			bBusy				=> xReadBusy,
			bError				=> xError,
			nErrID				=> udiErrID,
			iErrPos				=> usiErrPos,
			stMDP_DynAddr		=> ,
			iModuleTypeCount	=> ,
			iModuleCount		=> ,
			stMDP_ModuleHeader	=> ,
			arrStartIdx			=> ,
		);
	ELSE
		fbMDP_ReadModule(
			bExecute			:= FALSE,

			bBusy				=> xReadBusy,
			bError				=> xError,
			nErrID 				=> udiErrID,
			iErrPos				=> usiErrPos,
		);
		IF NOT xReadBusy THEN
			// allocate received module header
			stMDP_ModuleHeader	:= fbMDP_ReadModule.stMDP_ModuleHeader;
			// allocate information of startindexes in data buffer
			MEMCPY(ADR(arrStartIdx), ADR(fbMDP_ReadModule.arrStartIdx), SIZEOF(arrStartIdx) );
			// reset module content struct
			MEMSET( ADR(stMDP_ModuleContent), 0, SIZEOF(stMDP_ModuleContent) );
			// allocate received data to DiskMngmntTBL4 struct
			stMDP_ModuleContent.uiLen		:= arrData[0];
			MEMCPY(ADR(stMDP_ModuleContent.udiDriveType1), 	ADR(arrData)+arrStartIdx[1], MIN(arrStartIdx[2]-arrStartIdx[1], SIZEOF(stMDP_ModuleContent.udiDriveType1)) );
			MEMCPY(ADR(stMDP_ModuleContent.udiDriveType2), 	ADR(arrData)+arrStartIdx[2], MIN(arrStartIdx[3]-arrStartIdx[2], SIZEOF(stMDP_ModuleContent.udiDriveType2))  );
			MEMCPY(ADR(stMDP_ModuleContent.udiDriveType3), 	ADR(arrData)+arrStartIdx[3], MIN(arrStartIdx[4]-arrStartIdx[3], SIZEOF(stMDP_ModuleContent.udiDriveType3)) );
			MEMCPY(ADR(stMDP_ModuleContent.udiDriveType4), 	ADR(arrData)+arrStartIdx[4], MIN(arrStartIdx[5]-arrStartIdx[4], SIZEOF(stMDP_ModuleContent.udiDriveType4)) );
			MEMCPY(ADR(stMDP_ModuleContent.udiDriveType5),	ADR(arrData)+arrStartIdx[5], MIN(arrStartIdx[6]-arrStartIdx[5], SIZEOF(stMDP_ModuleContent.udiDriveType5)) );
			MEMCPY(ADR(stMDP_ModuleContent.udiDriveType6),	ADR(arrData)+arrStartIdx[6], MIN(arrStartIdx[7]-arrStartIdx[6], SIZEOF(stMDP_ModuleContent.udiDriveType6)) );

			// reset FB
			xBusy 				:= FALSE;
		END_IF
	END_IF

	// check timeout
	TimeOut();
	IF TimeOut.Q THEN
		TimeOut(IN 				:= FALSE);
		xError					:= TRUE;
		udiErrID				:= INT_TO_UINT(eMDP_Err_PLC) * 16#10000 + INT_TO_UINT(eMDP_ErrPLC_TimeOut);
	END_IF
END_IF

IF xError THEN
	// reset FB
	xBusy 						:= FALSE;
END_IF

END_FUNCTION_BLOCK

// ---- POUs/Safety_Diagnostics/AX5805_ADS_Reads.TcPOU
PROGRAM AX5805_ADS_Reads
//		8-2-2012
// 		This Program has been supplied by Beckhoff Automation As-Is and is intended only as an example 
//		implementation. Functionality is not guaranteed. 
//
VAR
	//Time to check CoE values
	T1							: 		TON ;
	xExecute					: 		BOOL ;
	tTime1						: 		TIME ;

	//Counter for just some very simple sequencing
	C1							: 		CTU ;
	xReset						: 		BOOL ;
	wPreset						: 		WORD := 10 ;
	xDone						: 		BOOL ;
	wCount						: 		WORD ;

	// Reading the serial number out of the AX5805
	fbAX5805Sn_ADSRead			: 		ADSREAD ;
	dwAX5805_Sn					: 		DWORD ;
	xAX5805Sn_busy				: 		BOOL ;
	xAX5805Sn_Err				: 		BOOL ;
	xAX5805Sn_ErrID				: 		UDINT ;

	// Reading the DIP Switch Setting out of the AX5805
	fbAX5805DSw_ADSRead			: 		ADSREAD ;
	wAX5805_DSw					: 		WORD ;
	xAX5805DSw_busy				: 		BOOL ;
	xAX5805DSw_Err				: 		BOOL ;
	udiAX5805DSw_ErrID			: 		UDINT ;

	//Read the Hardware Version of the AX5805 Logic Terminal
	fbAX5805_HWvers_EcCoESdoRead: 		FB_EcCoESdoRead ;
	sAX5805_HWvers				: 		STRING(2) ;
	xAX5805_HWvers_Busy			: 		BOOL ;
	xAX5805_HWvers_Err			: 		BOOL ;
	udiAX5805_HWvers_ErrID		: 		UDINT ;

	//Read the Software Version of the AX5805 Logic Terminal (It's f/w)
	fbAX5805_FWvers_EcCoESdoRead: 		FB_EcCoESdoRead ;
	sAX5805_FWvers				: 		STRING(2) ;
	xAX5805_FWvers_Busy			: 		BOOL ;
	xAX5805_FWvers_Err			: 		BOOL ;
	udiAX5805_FWvers_ErrID		: 		UDINT ;

	//Read the Number Of Connections Configured In The AX5805 Logic Terminal
	fbAX5805_StatConn_EcCoESdoRead: 	FB_EcCoESdoRead ;
	bAX5805_NoOfConnections		: 		BYTE ;
	xAX5805_NoOfConnections_Busy: 		BOOL ;
	xAX5805_NoOfConnections_Err	: 		BOOL ;
	udiAX5805_NoOfConnections_ErrID: 	UDINT ;

	//Read the Number Of Safety Groups Configured In The AX5805 Logic Terminal
	fbAX5805_SafetyGrps_EcCoESdoRead: 	FB_EcCoESdoRead ;
	bAX5805_NoOfSafetyGrps		: 		BYTE ;
	xAX5805_NoOfSafetyGrps_Busy	: 		BOOL ;
	xAX5805_NoOfSafetyGrps_Err	: 		BOOL ;
	udiAX5805_NoOfSafetyGrps_ErrID: 	UDINT ;

	//Read the Number Of Safety Function Blocks Configured In The AX5805 Logic Terminal
	fbAX5805_SafetyFBs_EcCoESdoRead: 	FB_EcCoESdoRead ;
	bAX5805_NoOfSafetyFBs		: 		BYTE ;
	xAX5805_NoOfSafetyFBs_Busy	: 		BOOL ;
	xAX5805_NoOfSafetyFBs_Err	: 		BOOL ;
	udiAX5805_NoOfSafetyFBs_ErrID: 		UDINT ;
	
	// Reading the Primary Micro Controller (MC1) Temperature in DegC out of the AX5805
	fbAX5805PriMCTemp_ADSRead	: 		ADSREAD ;
	wAX5805_PriMCTemp			: 		WORD ;
	xAX5805PriMCTemp_busy		: 		BOOL ;
	xAX5805PriMCTemp_Err		: 		BOOL ;
	udiAX5805PriMCTemp_ErrID	: 		UDINT ;

	// Reading the Secondary Micro Controller (MC2) Temperature in DegC out of the AX5805
	fbAX5805SecMCTemp_ADSRead	: 		ADSREAD ;
	wAX5805_SecMCTemp			: 		WORD ;
	xAX5805SecMCTemp_busy		: 		BOOL ;
	xAX5805SecMCTemp_Err		: 		BOOL ;
	udiAX5805SecMCTemp_ErrID	: 		UDINT ;

	// Reading the Primary Micro Controller (MC1) Voltage in mV out of the AX5805
	fbAX5805PriMC3300mV_ADSRead	: 		ADSREAD ;
	wAX5805_PriMC3300mV			: 		WORD ;
	xAX5805PriMC3300mV_busy		: 		BOOL ;
	xAX5805PriMC3300mV_Err		: 		BOOL ;
	udiAX5805PriMC3300mV_ErrID	: 		UDINT ;
	fbAX5805PriMC5000mV_ADSRead	: 		ADSREAD ;
	wAX5805_PriMC5000mV			: 		WORD ;
	xAX5805PriMC5000mV_busy		: 		BOOL ;
	xAX5805PriMC5000mV_Err		: 		BOOL ;
	udiAX5805PriMC5000mV_ErrID	: 		UDINT ;
	
	// Reading the Secondary Micro Controller (MC2) Voltage in mV out of the AX5805
	fbAX5805SecMC3300mV_ADSRead	: 		ADSREAD ;
	wAX5805_SecMC3300mV			: 		WORD ;
	xAX5805SecMC3300mV_busy		: 		BOOL ;
	xAX5805SecMC3300mV_Err		: 		BOOL ;
	udiAX5805SecMC3300mV_ErrID	: 		UDINT ;
	fbAX5805SecMC5000mV_ADSRead	: 		ADSREAD ;
	wAX5805_SecMC5000mV			: 		WORD ;
	xAX5805SecMC5000mV_busy		: 		BOOL ;
	xAX5805SecMC5000mV_Err		: 		BOOL ;
	udiAX5805SecMC5000mV_ErrID	: 		UDINT ;

	//Read the Configured Safety Option In The AX5000 Drive
	fbAX5000_SafetyOption				: 		FB_SoERead ;
	dwSafetyOption						: 		DWORD ;
	Axis1 								: 		AXIS_REF ;
	xAX5000_SafetyOption_busy			: 		BOOL ;
	xAX5000_SafetyOption_Err			: 		BOOL ;
	udiAX5000_SafetyOption_ErrID		: 		UDINT ;
	uiAX5000_SafetyOption_SercosErrID	: 		UINT ;
	dwAX5000_SafetyOption_Attribute		: 		DWORD ;
	
	//Read the Configured Motor String For CH-A in The AX5000 Drive
	fbAX5000_ConfigMotorCHA				: 		FB_SoERead ;
	sConfigMotorCHA						: 		STRING(30) ;
	xAX5000_sConfigMotorCHA_busy		: 		BOOL ;
	xAX5000_sConfigMotorCHA_Err			: 		BOOL ;
	udiAX5000_sConfigMotorCHA_ErrID		: 		UINT ;
	xAX5000_ConfigMotorCHA_busy			: 		BOOL ;
	xAX5000_ConfigMotorCHA_Err			:		BOOL ;
	udiAX5000_ConfigMotorCHA_ErrID		: 		UDINT ;
	uiAX5000_ConfigMotorCHA_SercosErrID	: 		UINT ;
	dwAX5000_ConfigMotorCHA_Attribute	: 		DWORD ;
	ConfigMotorCHA						: 		ARRAY[0..29] OF UINT ;
END_VAR
VAR_INPUT
END_VAR

//		8-2-2012
// 		This Program has been supplied by Beckhoff Automation As-Is and is intended only as an example 
//		implementation. Functionality is not guaranteed. 
//
IF g_bHMI_ScreenBeingDisplayed = 60 THEN
// Interval timer for CoE Reads
T1(
						IN				:= 		NOT xExecute, 
						PT				:=		T#500MS, 
						Q				=>		xExecute, 
						ET				=>		tTime1 ) ;

C1(
						CU				:= 		xExecute, 
						RESET			:= 		xReset, 
						PV				:= 		wPreset, 
						Q				=> 		xDone, 
						CV				=> 		wCount) ;

IF C1.CV > 6 	THEN xReset := 1 ;
				ELSE xReset := 0 ; 
END_IF ;

// Read the serial number out of the AX5805
fbAX5805Sn_ADSRead(
						NETID			:= 		gc_sADSNetID, 
						PORT			:= 		gc_uiAX5805_EtherCATAdr, 
						IDXGRP			:= 		16#F302, 
						IDXOFFS			:= 		16#F9800002, 
						LEN				:= 		4, 
						DESTADDR		:= 		ADR(dwAX5805_Sn), 
						READ			:= 		xExecute, 
						TMOUT			:= 		T#2S, 
						BUSY			=> 		xAX5805Sn_busy, 
						ERR				=> 		xAX5805Sn_Err, 
						ERRID			=> 		xAX5805Sn_ErrID );

g_dwHMI_AX5805Sn 						:= 		dwAX5805_Sn ;

// Read the DIP Switch Setting out of the AX5805
IF C1.CV = 1 THEN
fbAX5805DSw_ADSRead(
						NETID			:= 		gc_sADSNetID, 
						PORT			:= 		gc_uiAX5805_EtherCATAdr, 
						IDXGRP			:= 		16#F302, 
						IDXOFFS			:= 		16#F9800001, 
						LEN				:= 		2, 
						DESTADDR		:= 		ADR(wAX5805_DSw), 
						READ			:= 		xExecute, 
						TMOUT			:= 		T#2S, 
						BUSY			=> 		xAX5805DSw_busy, 
						ERR				=> 		xAX5805DSw_Err, 
						ERRID			=> 		udiAX5805DSw_ErrID );

g_wHMI_AX5805DSw 						:= 		wAX5805_DSw ;
END_IF ;						

//Read the Hardware Version of the AX5805 Logic Terminal
fbAX5805_HWvers_EcCoESdoRead(
						sNetId			:= 		gc_sADSNetID, 
						nSlaveAddr		:= 		gc_uiAX5805_EtherCATAdr, 
						nSubIndex		:= 		0, 
						nIndex			:= 		16#1009, 
						pDstBuf			:=  	ADR(sAX5805_HWvers),
						cbBufLen		:= 		SIZEOF(sAX5805_HWvers), 
						bExecute		:= 		xExecute, 
						tTimeout		:= 		T#2S, 
						bBusy			=> 		xAX5805_HWvers_Busy, 
						bError			=> 		xAX5805_HWvers_Err, 
						nErrId			=> 		udiAX5805_HWvers_ErrID ) ;

g_sHMI_AX5805_HWvers					:= 		sAX5805_HWvers ;

//Read the Software Version of the AX5805 Logic Terminal (It's f/w)
fbAX5805_FWvers_EcCoESdoRead(
						sNetId			:= 		gc_sADSNetID, 
						nSlaveAddr		:= 		gc_uiAX5805_EtherCATAdr, 
						nSubIndex		:= 		0, 
						nIndex			:= 		16#100A, 
						pDstBuf			:=  	ADR(sAX5805_FWvers),
						cbBufLen		:= 		SIZEOF(sAX5805_FWvers), 
						bExecute		:= 		xExecute, 
						tTimeout		:= 		T#2S, 
						bBusy			=> 		xAX5805_FWvers_Busy, 
						bError			=> 		xAX5805_FWvers_Err, 
						nErrId			=> 		udiAX5805_FWvers_ErrID ) ;

g_sHMI_AX5805_FWvers					:= 		sAX5805_FWvers ;

// Read the Primary Micro Controller (MC1) Temperature in DegC out of the AX5805
IF C1.CV = 2 THEN
fbAX5805PriMCTemp_ADSRead(
						NETID			:= 		gc_sADSNetID, 
						PORT			:= 		gc_uiAX5805_EtherCATAdr, 
						IDXGRP			:= 		16#F302, 
						IDXOFFS			:= 		16#FA800001, 
						LEN				:= 		2, 
						DESTADDR		:= 		ADR(wAX5805_PriMCTemp), 
						READ			:= 		xExecute, 
						TMOUT			:= 		T#2S, 
						BUSY			=> 		xAX5805PriMCTemp_busy, 
						ERR				=> 		xAX5805PriMCTemp_Err, 
						ERRID			=> 		udiAX5805PriMCTemp_ErrID );

g_wHMI_AX5805PriMCTemp 					:= 		wAX5805_PriMCTemp ;
END_IF ;

// Read the Secondary Micro Controller (MC2) Temperature in DegC out of the AX5805
IF C1.CV = 3 THEN
fbAX5805SecMCTemp_ADSRead(
						NETID			:= 		gc_sADSNetID, 
						PORT			:= 		gc_uiAX5805_EtherCATAdr, 
						IDXGRP			:= 		16#F302, 
						IDXOFFS			:= 		16#FA800002, 
						LEN				:= 		2, 
						DESTADDR		:= 		ADR(wAX5805_SecMCTemp), 
						READ			:= 		xExecute, 
						TMOUT			:= 		T#2S, 
						BUSY			=> 		xAX5805SecMCTemp_busy, 
						ERR				=> 		xAX5805SecMCTemp_Err, 
						ERRID			=> 		udiAX5805SecMCTemp_ErrID );

g_wHMI_AX5805SecMCTemp 					:= 		wAX5805_SecMCTemp ;
END_IF ;

// Read the Primary Micro Controller (MC1) 3.3v Nominal Voltage in mV out of the AX5805
IF C1.CV = 4 THEN
fbAX5805PriMC3300mV_ADSRead(
						NETID			:= 		gc_sADSNetID, 
						PORT			:= 		gc_uiAX5805_EtherCATAdr, 
						IDXGRP			:= 		16#F302, 
						IDXOFFS			:= 		16#FA810001, 
						LEN				:= 		2, 
						DESTADDR		:= 		ADR(wAX5805_PriMC3300mV), 
						READ			:= 		xExecute, 
						TMOUT			:= 		T#2S, 
						BUSY			=> 		xAX5805PriMC3300mV_busy, 
						ERR				=> 		xAX5805PriMC3300mV_Err, 
						ERRID			=> 		udiAX5805PriMC3300mV_ErrID );

g_wHMI_AX5805PriMC_3p3Volts				:= 		WORD_TO_LREAL(wAX5805_PriMC3300mV) / 1000.0 ;
END_IF ;

// Read the Secondary Micro Controller (MC2) 3.3v Nominal Voltage in mV out of the AX5805
IF C1.CV = 5 THEN
fbAX5805SecMC3300mV_ADSRead(
						NETID			:= 		gc_sADSNetID, 
						PORT			:= 		gc_uiAX5805_EtherCATAdr, 
						IDXGRP			:= 		16#F302, 
						IDXOFFS			:= 		16#FA810002, 
						LEN				:= 		2, 
						DESTADDR		:= 		ADR(wAX5805_SecMC3300mV), 
						READ			:= 		xExecute, 
						TMOUT			:= 		T#2S, 
						BUSY			=> 		xAX5805SecMC3300mV_busy, 
						ERR				=> 		xAX5805SecMC3300mV_Err, 
						ERRID			=> 		udiAX5805SecMC3300mV_ErrID );
			
g_wHMI_AX5805SecMC_3p3Volts 				:= 		WORD_TO_LREAL(wAX5805_SecMC3300mV) / 1000.0 ;
END_IF ;

// Read the Primary Micro Controller (MC1) 5.0v Nominal Voltage in mV out of the AX5805
IF C1.CV = 1 THEN
fbAX5805PriMC5000mV_ADSRead(
						NETID			:= 		gc_sADSNetID, 
						PORT			:= 		gc_uiAX5805_EtherCATAdr, 
						IDXGRP			:= 		16#F302, 
						IDXOFFS			:= 		16#FA810003, 
						LEN				:= 		2, 
						DESTADDR		:= 		ADR(wAX5805_PriMC5000mV), 
						READ			:= 		xExecute, 
						TMOUT			:= 		T#2S, 
						BUSY			=> 		xAX5805PriMC5000mV_busy, 
						ERR				=> 		xAX5805PriMC5000mV_Err, 
						ERRID			=> 		udiAX5805PriMC5000mV_ErrID );

g_wHMI_AX5805PriMC_5Volts				:= 		WORD_TO_LREAL(wAX5805_PriMC5000mV) / 1000.0 ;
END_IF ;

// Read the Secondary Micro Controller (MC2) 5.0v Nominal Voltage in mV out of the AX5805
IF C1.CV = 2 THEN
fbAX5805SecMC5000mV_ADSRead(
						NETID			:= 		gc_sADSNetID, 
						PORT			:= 		gc_uiAX5805_EtherCATAdr, 
						IDXGRP			:= 		16#F302, 
						IDXOFFS			:= 		16#FA810004, 
						LEN				:= 		2, 
						DESTADDR		:= 		ADR(wAX5805_SecMC5000mV), 
						READ			:= 		xExecute, 
						TMOUT			:= 		T#2S, 
						BUSY			=> 		xAX5805SecMC5000mV_busy, 
						ERR				=> 		xAX5805SecMC5000mV_Err, 
						ERRID			=> 		udiAX5805SecMC5000mV_ErrID );
			
g_wHMI_AX5805SecMC_5Volts 				:= 		WORD_TO_LREAL(wAX5805_SecMC5000mV) / 1000.0 ;
END_IF ;

(* Read the Configured Safety Option For CH-A in The AX5000 Drive

An advantage of using the FB_SoERead function block Form the MC2_Drive library
is the NedID is the controller's NetID not the EtherCAT master so it is possible 
to leave that field with just blank single quotes '' and the TwinCAT system 
assumes the NetID of the computer for you.

The MC2_Drive library has dependencies on the MC2 library in TwinCAT and Tc3 at this point
(build 3099.1) doesn't notice the dependancy and add the extra library for you.  You must
manually add it yourself.

	S_0_IDN		: WORD	:= 16#0000;
	S_1_IDN		: WORD	:= 16#1000;
	S_2_IDN		: WORD	:= 16#2000;
	S_3_IDN		: WORD	:= 16#3000;
	S_4_IDN		: WORD	:= 16#4000;
	S_5_IDN		: WORD	:= 16#5000;
	S_6_IDN		: WORD	:= 16#6000;
	S_7_IDN		: WORD	:= 16#7000;

	P_0_IDN		: WORD	:= 16#8000;
	P_1_IDN		: WORD	:= 16#9000;
	P_2_IDN		: WORD	:= 16#A000;
	P_3_IDN		: WORD	:= 16#B000;
	P_4_IDN		: WORD	:= 16#C000;
	P_5_IDN		: WORD	:= 16#D000;
	P_6_IDN		: WORD	:= 16#E000;
	P_7_IDN		: WORD	:= 16#F000;

A Few documented SERCOS error codes:
---------------------------------------
0x1003 Wrong parameter mode 
0x1004 Data parameter wrong value size 
0x1005 False backup parameter type  
0x1006 Backup list was not IDN 192 

nElement: Element number of the parameter that is to be written. The following values are allowed:
--------------------------------------------------------------------------------------------------
Value Description 
0x01 Data Status 
0x02 Name (read only) 
0x04 Attribute 
0x08 Unit 
0x10 Minimum 
0x20 Maximum 
0x40 Value 
0x80 Default 

*)
fbAX5000_SafetyOption(
						NetId			:= 		'', 
						Idn				:= 		DINT_TO_WORD(16#8000 + 2000), 
						Element			:= 		16#40, 
						pDstBuf			:= 		ADR(dwSafetyOption), 
						BufLen			:= 		SIZEOF(dwSafetyOption), 
						Execute			:= 		xExecute, 
						Timeout			:= 		T#2S, 
						Axis			:= 		Axis1, 
						Busy			=> 		xAX5000_SafetyOption_busy, 
						Error			=> 		xAX5000_SafetyOption_Err, 
						AdsErrId		=> 		udiAX5000_SafetyOption_ErrID, 
						SercosErrId		=> 		uiAX5000_SafetyOption_SercosErrID, 
						Attribute		=> 		dwAX5000_SafetyOption_Attribute) ;

IF dwSafetyOption 						= 		0 THEN
	g_sHMI_AX5000_SafetyOption			:= 		'No Safety Option Selected' ;
	ELSIF dwSafetyOption				= 		1 THEN
	g_sHMI_AX5000_SafetyOption			:= 		'AX5801 Option Selected' ;
	ELSIF dwSafetyOption				= 		2 THEN
	g_sHMI_AX5000_SafetyOption			:= 		'AX5805 Option Selected' ;
ELSE
	g_sHMI_AX5000_SafetyOption			:= 		'Invalid Option' ;
END_IF ;

//AX5000 Ch-A Motor String
fbAX5000_ConfigMotorCHA(
						NetId			:= 		'', 
						Idn				:= 		DINT_TO_WORD(16#8000 + 53), 
						Element			:= 		16#40, 
						pDstBuf			:= 		ADR(ConfigMotorCHA), 
						BufLen			:= 		SIZEOF(ConfigMotorCHA), 
						Execute			:= 		xExecute, 
						Timeout			:= 		T#2S, 
						Axis			:= 		Axis1, 
						Busy			=> 		xAX5000_ConfigMotorCHA_busy, 
						Error			=> 		xAX5000_ConfigMotorCHA_Err, 
						AdsErrId		=> 		udiAX5000_ConfigMotorCHA_ErrID, 
						SercosErrId		=> 		uiAX5000_ConfigMotorCHA_SercosErrID, 
						Attribute		=> 		dwAX5000_ConfigMotorCHA_Attribute) ;

g_sHMI_AX5000_ConfigMotorCHA 			:= 		 UINT_TO_STRING(ConfigMotorCHA[2]) ;

ELSE xReset := 1 ;
END_IF ;

END_PROGRAM

// ---- POUs/Safety_Diagnostics/EL6930_ADS_Reads.TcPOU
PROGRAM EL6930_ADS_Reads
//		8-2-2012
// 		This Program has been supplied by Beckhoff Automation As-Is and is intended only as an example 
//		implementation. Functionality is not guaranteed. 
//
VAR
	//Time to check CoE values
	T1							: 		TON ;
	xExecute					: 		BOOL ;
	tTime1						: 		TIME ;

	//Counter for just some very simple sequencing
	C1							: 		CTU ;
	xReset						: 		BOOL ;
	wPreset						: 		WORD := 10 ;
	xDone						: 		BOOL ;
	wCount						: 		WORD ;

	//Read the serial number out of the EL6930
	fbEL6930Sn_ADSRead			: 		ADSREAD ;
	dwEL6930_Sn					: 		DWORD ;
	xEL6930Sn_busy				: 		BOOL ;
	xEL6930Sn_Err				: 		BOOL ;
	xEL6930Sn_ErrID				: 		UDINT ;

	//Read the DIP Switch Setting out of the EL6930
	fbEL6930DSw_ADSRead			: 		ADSREAD ;
	wEL6930_DSw					: 		WORD ;
	xEL6930DSw_busy				: 		BOOL ;
	xEL6930DSw_Err				: 		BOOL ;
	udiEL6930DSw_ErrID			: 		UDINT ;

	//Read the Hardware Version of the EL6930 Logic Terminal
	fbEL6930_HWvers_EcCoESdoRead: 		FB_EcCoESdoRead ;
	sEL6930_HWvers				: 		STRING(2) ;
	xEL6930_HWvers_Busy			: 		BOOL ;
	xEL6930_HWvers_Err			: 		BOOL ;
	udiEL6930_HWvers_ErrID		: 		UDINT ;

	//Read the Software Version of the EL6930 Logic Terminal (It's f/w)
	fbEL6930_FWvers_EcCoESdoRead: 		FB_EcCoESdoRead ;
	sEL6930_FWvers				: 		STRING(2) ;
	xEL6930_FWvers_Busy			: 		BOOL ;
	xEL6930_FWvers_Err			: 		BOOL ;
	udiEL6930_FWvers_ErrID		: 		UDINT ;

	//Read the Number Of Connections Configured In The EL6930 Logic Terminal
	fbEL6930_StatConn_EcCoESdoRead: 	FB_EcCoESdoRead ;
	bNoOfConnections			: 		BYTE ;
	bEL6930_NoOfConnections		: 		BYTE ;
	xEL6930_NoOfConnections_Busy: 		BOOL ;
	xEL6930_NoOfConnections_Err	: 		BOOL ;
	udiEL6930_NoOfConnections_ErrID: 	UDINT ;

	//Read the Number Of Safety Groups Configured In The EL6930 Logic Terminal
	fbEL6930_SafetyGrps_EcCoESdoRead: 	FB_EcCoESdoRead ;
	bEL6930_NoOfSafetyGrps		: 		BYTE ;
	xEL6930_NoOfSafetyGrps_Busy	: 		BOOL ;
	xEL6930_NoOfSafetyGrps_Err	: 		BOOL ;
	udiEL6930_NoOfSafetyGrps_ErrID: 	UDINT ;

	//Read the Number Of Safety Function Blocks Configured In The EL6930 Logic Terminal
	fbEL6930_SafetyFBs_EcCoESdoRead: 	FB_EcCoESdoRead ;
	bEL6930_NoOfSafetyFBs		: 		BYTE ;
	xEL6930_NoOfSafetyFBs_Busy	: 		BOOL ;
	xEL6930_NoOfSafetyFBs_Err	: 		BOOL ;
	udiEL6930_NoOfSafetyFBs_ErrID: 		UDINT ;
	
	//Read the Primary Micro Controller (MC1) Temperature in DegC out of the EL6930
	fbEL6930PriMCTemp_ADSRead	: 		ADSREAD ;
	wEL6930_PriMCTemp			: 		WORD ;
	xEL6930PriMCTemp_busy		: 		BOOL ;
	xEL6930PriMCTemp_Err		: 		BOOL ;
	udiEL6930PriMCTemp_ErrID	: 		UDINT ;

	//Read the Secondary Micro Controller (MC2) Temperature in DegC out of the EL6930
	fbEL6930SecMCTemp_ADSRead	: 		ADSREAD ;
	wEL6930_SecMCTemp			: 		WORD ;
	xEL6930SecMCTemp_busy		: 		BOOL ;
	xEL6930SecMCTemp_Err		: 		BOOL ;
	udiEL6930SecMCTemp_ErrID	: 		UDINT ;

	//Read the Primary Micro Controller (MC1) Voltage in mV out of the EL6930
	fbEL6930PriMCmV_ADSRead		: 		ADSREAD ;
	wEL6930_PriMCmV				: 		WORD ;
	xEL6930PriMCmV_busy			: 		BOOL ;
	xEL6930PriMCmV_Err			: 		BOOL ;
	udiEL6930PriMCmV_ErrID		: 		UDINT ;

	//Read the Secondary Micro Controller (MC2) Voltage in mV out of the EL6930
	fbEL6930SecMCmV_ADSRead		: 		ADSREAD ;
	wEL6930_SecMCmV				: 		WORD ;
	xEL6930SecMCmV_busy			: 		BOOL ;
	xEL6930SecMCmV_Err			: 		BOOL ;
	udiEL6930SecMCmV_ErrID		: 		UDINT ;

	// EL6930: Temperature and Voltage Errors
	//There are two temperature sensors inside each Microcontroller
	fbEL6930_Error_ADSRead		: 		ADSREAD ;
	wEL6930_Error				: 		WORD ;
	xEL6930Error_busy			: 		BOOL ;
	xEL6930Error_Err			: 		BOOL ;
	udiEL6930Error_ErrID		: 		UDINT ;
END_VAR
VAR_INPUT
END_VAR

//		8-2-2012
// 		This Program has been supplied by Beckhoff Automation As-Is and is intended only as an example 
//		implementation. Functionality is not guaranteed. 
//
IF g_bHMI_ScreenBeingDisplayed = 50 THEN
// Interval timer for CoE Reads
T1(
						IN				:= 		NOT xExecute, 
						PT				:=		T#500MS, 
						Q				=>		xExecute, 
						ET				=>		tTime1 ) ;

C1(
						CU				:= 		xExecute, 
						RESET			:= 		xReset, 
						PV				:= 		wPreset, 
						Q				=> 		xDone, 
						CV				=> 		wCount) ;

IF C1.CV > 6 	THEN xReset := 1 ;
				ELSE xReset := 0 ; 
END_IF ;

// Read the serial number out of the EL6930
fbEL6930Sn_ADSRead(
						NETID			:= 		gc_sADSNetID, 
						PORT			:= 		gc_uiEL6930_EtherCATAdr, 
						IDXGRP			:= 		16#F302, 
						IDXOFFS			:= 		16#F9800002, 
						LEN				:= 		4, 
						DESTADDR		:= 		ADR(dwEL6930_Sn), 
						READ			:= 		xExecute, 
						TMOUT			:= 		T#2S, 
						BUSY			=> 		xEL6930Sn_busy, 
						ERR				=> 		xEL6930Sn_Err, 
						ERRID			=> 		xEL6930Sn_ErrID );

g_dwHMI_EL6930Sn 						:= 		dwEL6930_Sn ;

// Read the DIP Switch Setting out of the EL6930
IF C1.CV = 1 THEN
fbEL6930DSw_ADSRead(
						NETID			:= 		gc_sADSNetID, 
						PORT			:= 		gc_uiEL6930_EtherCATAdr, 
						IDXGRP			:= 		16#F302, 
						IDXOFFS			:= 		16#F9800001, 
						LEN				:= 		2, 
						DESTADDR		:= 		ADR(wEL6930_DSw), 
						READ			:= 		xExecute, 
						TMOUT			:= 		T#2S, 
						BUSY			=> 		xEL6930DSw_busy, 
						ERR				=> 		xEL6930DSw_Err, 
						ERRID			=> 		udiEL6930DSw_ErrID );

g_wHMI_EL6930DSw 						:= 		wEL6930_DSw ;
END_IF ;						

//Read the Hardware Version of the EL6930 Logic Terminal
fbEL6930_HWvers_EcCoESdoRead(
						sNetId			:= 		gc_sADSNetID, 
						nSlaveAddr		:= 		gc_uiEL6930_EtherCATAdr, 
						nSubIndex		:= 		0, 
						nIndex			:= 		16#1009, 
						pDstBuf			:=  	ADR(sEL6930_HWvers),
						cbBufLen		:= 		SIZEOF(sEL6930_HWvers), 
						bExecute		:= 		xExecute, 
						tTimeout		:= 		T#2S, 
						bBusy			=> 		xEL6930_HWvers_Busy, 
						bError			=> 		xEL6930_HWvers_Err, 
						nErrId			=> 		udiEL6930_HWvers_ErrID ) ;

g_sHMI_EL6930_HWvers					:= 		sEL6930_HWvers ;

//Read the Software Version of the EL6930 Logic Terminal (It's f/w)
fbEL6930_FWvers_EcCoESdoRead(
						sNetId			:= 		gc_sADSNetID, 
						nSlaveAddr		:= 		gc_uiEL6930_EtherCATAdr, 
						nSubIndex		:= 		0, 
						nIndex			:= 		16#100A, 
						pDstBuf			:=  	ADR(sEL6930_FWvers),
						cbBufLen		:= 		SIZEOF(sEL6930_FWvers), 
						bExecute		:= 		xExecute, 
						tTimeout		:= 		T#2S, 
						bBusy			=> 		xEL6930_FWvers_Busy, 
						bError			=> 		xEL6930_FWvers_Err, 
						nErrId			=> 		udiEL6930_FWvers_ErrID ) ;

g_sHMI_EL6930_FWvers					:= 		sEL6930_FWvers ;

//Read the Number Of Connections Configured In The EL6930 Logic Terminal
fbEL6930_StatConn_EcCoESdoRead(
						sNetId			:= 		gc_sADSNetID, 
						nSlaveAddr		:= 		gc_uiEL6930_EtherCATAdr, 
						nSubIndex		:= 		0, 
						nIndex			:= 		16#2110, 
						pDstBuf			:=  	ADR(bEL6930_NoOfConnections),
						cbBufLen		:= 		SIZEOF(bEL6930_NoOfConnections), 
						bExecute		:= 		xExecute, 
						tTimeout		:= 		T#2S, 
						bBusy			=> 		xEL6930_NoOfConnections_Busy, 
						bError			=> 		xEL6930_NoOfConnections_Err, 
						nErrId			=> 		udiEL6930_NoOfConnections_ErrID ) ;

g_bHMI_EL6930_NoOfConnections			:= 		bEL6930_NoOfConnections ;					

//Read the Number Of Safety Groups Configured In The EL6930 Logic Terminal
fbEL6930_SafetyGrps_EcCoESdoRead(
						sNetId			:= 		gc_sADSNetID, 
						nSlaveAddr		:= 		gc_uiEL6930_EtherCATAdr, 
						nSubIndex		:= 		0, 
						nIndex			:= 		16#2120, 
						pDstBuf			:=  	ADR(bEL6930_NoOfSafetyGrps),
						cbBufLen		:= 		SIZEOF(bEL6930_NoOfSafetyGrps), 
						bExecute		:= 		xExecute, 
						tTimeout		:= 		T#2S, 
						bBusy			=> 		xEL6930_NoOfSafetyGrps_Busy, 
						bError			=> 		xEL6930_NoOfSafetyGrps_Err, 
						nErrId			=> 		udiEL6930_NoOfSafetyGrps_ErrID ) ;

g_bHMI_EL6930_NoOfSafetyGrps			:= 		bEL6930_NoOfSafetyGrps ;

//Read the Number Of Safety Function Blocks Configured In The EL6930 Logic Terminal
fbEL6930_SafetyFBs_EcCoESdoRead(
						sNetId			:= 		gc_sADSNetID, 
						nSlaveAddr		:= 		gc_uiEL6930_EtherCATAdr, 
						nSubIndex		:= 		0, 
						nIndex			:= 		16#2130, 
						pDstBuf			:=  	ADR(bEL6930_NoOfSafetyFBs),
						cbBufLen		:= 		SIZEOF(bEL6930_NoOfSafetyFBs), 
						bExecute		:= 		xExecute, 
						tTimeout		:= 		T#2S, 
						bBusy			=> 		xEL6930_NoOfSafetyFBs_Busy, 
						bError			=> 		xEL6930_NoOfSafetyFBs_Err, 
						nErrId			=> 		udiEL6930_NoOfSafetyFBs_ErrID ) ;

g_bHMI_EL6930_NoOfSafetyFBs			:= 		bEL6930_NoOfSafetyFBs ;

// Read the Primary Micro Controller (MC1) Temperature in DegC out of the EL6930
IF C1.CV = 2 THEN
fbEL6930PriMCTemp_ADSRead(
						NETID			:= 		gc_sADSNetID, 
						PORT			:= 		gc_uiEL6930_EtherCATAdr, 
						IDXGRP			:= 		16#F302, 
						IDXOFFS			:= 		16#FA800001, 
						LEN				:= 		2, 
						DESTADDR		:= 		ADR(wEL6930_PriMCTemp), 
						READ			:= 		xExecute, 
						TMOUT			:= 		T#2S, 
						BUSY			=> 		xEL6930PriMCTemp_busy, 
						ERR				=> 		xEL6930PriMCTemp_Err, 
						ERRID			=> 		udiEL6930PriMCTemp_ErrID );

g_wHMI_EL6930PriMCTemp 						:= 		wEL6930_PriMCTemp ;
END_IF ;

// Read the Secondary Micro Controller (MC2) Temperature in DegC out of the EL6930
IF C1.CV = 3 THEN
fbEL6930SecMCTemp_ADSRead(
						NETID			:= 		gc_sADSNetID, 
						PORT			:= 		gc_uiEL6930_EtherCATAdr, 
						IDXGRP			:= 		16#F302, 
						IDXOFFS			:= 		16#FA800002, 
						LEN				:= 		2, 
						DESTADDR		:= 		ADR(wEL6930_SecMCTemp), 
						READ			:= 		xExecute, 
						TMOUT			:= 		T#2S, 
						BUSY			=> 		xEL6930SecMCTemp_busy, 
						ERR				=> 		xEL6930SecMCTemp_Err, 
						ERRID			=> 		udiEL6930SecMCTemp_ErrID );

g_wHMI_EL6930SecMCTemp 						:= 		wEL6930_SecMCTemp ;
END_IF ;

// Read the Primary Micro Controller (MC1) Voltage in mV out of the EL6930
IF C1.CV = 4 THEN
fbEL6930PriMCmV_ADSRead(
						NETID			:= 		gc_sADSNetID, 
						PORT			:= 		gc_uiEL6930_EtherCATAdr, 
						IDXGRP			:= 		16#F302, 
						IDXOFFS			:= 		16#FA800003, 
						LEN				:= 		2, 
						DESTADDR		:= 		ADR(wEL6930_PriMCmV), 
						READ			:= 		xExecute, 
						TMOUT			:= 		T#2S, 
						BUSY			=> 		xEL6930PriMCmV_busy, 
						ERR				=> 		xEL6930PriMCmV_Err, 
						ERRID			=> 		udiEL6930PriMCmV_ErrID );

g_wHMI_EL6930PriMC_Volts				:= 		WORD_TO_LREAL(wEL6930_PriMCmV) / 1000.0 ;
END_IF ;

// Read the Secondary Micro Controller (MC2) Voltage in mV out of the EL6930
IF C1.CV = 5 THEN
fbEL6930SecMCmV_ADSRead(
						NETID			:= 		gc_sADSNetID, 
						PORT			:= 		gc_uiEL6930_EtherCATAdr, 
						IDXGRP			:= 		16#F302, 
						IDXOFFS			:= 		16#FA800004, 
						LEN				:= 		2, 
						DESTADDR		:= 		ADR(wEL6930_SecMCmV), 
						READ			:= 		xExecute, 
						TMOUT			:= 		T#2S, 
						BUSY			=> 		xEL6930SecMCmV_busy, 
						ERR				=> 		xEL6930SecMCmV_Err, 
						ERRID			=> 		udiEL6930SecMCmV_ErrID );
			
g_wHMI_EL6930SecMC_Volts 				:= 		WORD_TO_LREAL(wEL6930_SecMCmV) / 1000.0 ;
END_IF ;
	ELSE xReset := 1 ;
	END_IF ;

//EL6930: Temperature and Voltage Errors
//There are two temperature sensors inside each Microcontroller
fbEL6930_Error_ADSRead(
						NETID			:= 		gc_sADSNetID, 
						PORT			:= 		gc_uiEL6930_EtherCATAdr, 
						IDXGRP			:= 		16#F302, 
						IDXOFFS			:= 		16#FA000003, 
						LEN				:= 		2, 
						DESTADDR		:= 		ADR(wEL6930_Error), 
						READ			:= 		xExecute, 
						TMOUT			:= 		T#2S, 
						BUSY			=> 		xEL6930Error_busy, 
						ERR				=> 		xEL6930Error_Err, 
						ERRID			=> 		udiEL6930Error_ErrID );
			
//These errors may only be present temporarily so they need to be latched and then cleared
//to be properly noted by the operator
g_xHMI_EL6930_MaxTemp				:= 		(wEL6930_Error = 5) OR (g_xHMI_EL6930_MaxTemp AND NOT g_xHMI_EL6930_ErrClearPB) ;
g_xHMI_EL6930_MinTemp				:= 		(wEL6930_Error = 6) OR (g_xHMI_EL6930_MinTemp AND NOT g_xHMI_EL6930_ErrClearPB) ;
g_xHMI_EL6930_TempDiffExceeded		:= 		(wEL6930_Error = 7) OR (g_xHMI_EL6930_TempDiffExceeded AND NOT g_xHMI_EL6930_ErrClearPB) ;
g_xHMI_EL6930_MaxVccMC1				:= 		(wEL6930_Error = 257) OR (g_xHMI_EL6930_MaxVccMC1 AND NOT g_xHMI_EL6930_ErrClearPB) ;
g_xHMI_EL6930_MaxVccMC2				:= 		(wEL6930_Error = 258) OR (g_xHMI_EL6930_MaxVccMC2 AND NOT g_xHMI_EL6930_ErrClearPB) ;
g_xHMI_EL6930_MinVccMC1				:= 		(wEL6930_Error = 259) OR (g_xHMI_EL6930_MinVccMC1 AND NOT g_xHMI_EL6930_ErrClearPB) ;
g_xHMI_EL6930_MinVccMC2				:= 		(wEL6930_Error = 260) OR (g_xHMI_EL6930_MinVccMC2 AND NOT g_xHMI_EL6930_ErrClearPB) ;

//Sum of all errors we know of in the EL6930 terminal
IF 		g_xHMI_EL6930_MaxTemp 
	OR 	g_xHMI_EL6930_MinTemp
	OR 	g_xHMI_EL6930_TempDiffExceeded 
	OR 	g_xHMI_EL6930_MaxVccMC1
	OR 	g_xHMI_EL6930_MaxVccMC2
	OR 	g_xHMI_EL6930_MinVccMC1
	OR 	g_xHMI_EL6930_MinVccMC2
		THEN g_xHMI_EL6930_General_Error := TRUE ;
		ELSE g_xHMI_EL6930_General_Error := FALSE ;
END_IF ;

END_PROGRAM

// ---- POUs/Safety_Diagnostics/EP1908_ADS_Reads.TcPOU
PROGRAM EP1908_ADS_Reads
VAR
//		8-2-2012
// 		This Program has been supplied by Beckhoff Automation As-Is and is intended only as an example 
//		implementation. Functionality is not guaranteed. 
//
	//Time to check CoE values (Every 2 seconds in this case)
	T1							: 		TON ;
	xExecute					: 		BOOL ;
	tTime1						: 		TIME ;

	//Counter for just some very simple sequencing
	C1							: 		CTU ;
	xReset						: 		BOOL ;
	wPreset						: 		WORD := 10 ;
	xDone						: 		BOOL ;
	wCount						: 		WORD ;

	// Reading the serial number out of the EP1908-0002
	fbEP1908Sn_ADSRead			: 		ADSREAD ;
	dwEP1908_Sn					: 		DWORD ;
	xEP1908Sn_busy				: 		BOOL ;
	xEP1908Sn_Err				: 		BOOL ;
	xEP1908Sn_ErrID				: 		UDINT ;

	// Reading the DIP Switch Setting out of the EP1908-0002
	fbEP1908DSw_ADSRead			: 		ADSREAD ;
	wEP1908_DSw					: 		WORD ;
	xEP1908DSw_busy				: 		BOOL ;
	xEP1908DSw_Err				: 		BOOL ;
	udiEP1908DSw_ErrID			: 		UDINT ;

	//Read the Hardware Version of the EP1908-0002 Terminal
	fbEP1908_HWvers_EcCoESdoRead	: 	FB_EcCoESdoRead ;
	sEP1908_HWvers					: 	STRING(2) ;
	xEP1908_HWvers_Busy				: 	BOOL ;
	xEP1908_HWvers_Err				: 	BOOL ;
	udiEP1908_HWvers_ErrID			: 	UDINT ;

	//Read the Software Version of the EP1908-0002 Logic Terminal (It's f/w)
	fbEP1908_FWvers_EcCoESdoRead	: 	FB_EcCoESdoRead ;
	sEP1908_FWvers					: 	STRING(2) ;
	xEP1908_FWvers_Busy				: 	BOOL ;
	xEP1908_FWvers_Err				: 	BOOL ;
	udiEP1908_FWvers_ErrID			: 	UDINT ;
	
	// Reading the Primary Micro Controller (MC1) Temperature in DegC out of the EP1908-0002
	fbEP1908PriMCTemp_ADSRead	: 		ADSREAD ;
	wEP1908_PriMCTemp			: 		WORD ;
	xEP1908PriMCTemp_busy		: 		BOOL ;
	xEP1908PriMCTemp_Err		: 		BOOL ;
	udiEP1908PriMCTemp_ErrID	: 		UDINT ;

	// Reading the Secondary Micro Controller (MC2) Temperature in DegC out of the EP1908-0002
	fbEP1908SecMCTemp_ADSRead	: 		ADSREAD ;
	wEP1908_SecMCTemp			: 		WORD ;
	xEP1908SecMCTemp_busy		: 		BOOL ;
	xEP1908SecMCTemp_Err		: 		BOOL ;
	udiEP1908SecMCTemp_ErrID	: 		UDINT ;

	// Reading the Primary Micro Controller (MC1) Voltage in mV out of the EP1908-0002
	fbEP1908PriMCmV_ADSRead		: 		ADSREAD ;
	wEP1908_PriMCmV				: 		WORD ;
	xEP1908PriMCmV_busy			: 		BOOL ;
	xEL1904PriMCmV_Err			: 		BOOL ;
	xEP1908PriMCmV_Err			: 		BOOL ;
	udiEP1908PriMCmV_ErrID		: 		UDINT ;

	// Reading the Secondary Micro Controller (MC2) Voltage in mV out of the EP1908-0002
	fbEP1908SecMCmV_ADSRead		: 		ADSREAD ;
	wEP1908_SecMCmV				: 		WORD ;
	xEP1908SecMCmV_busy			: 		BOOL ;
	xEP1908SecMCmV_Err			: 		BOOL ;
	udiEP1908SecMCmV_ErrID		: 		UDINT ;

	// EP1908-0002: Sensor Test Error
	fbEP1908SensT_ADSRead		: 		ADSREAD ;
	wEP1908_SenT				: 		WORD ;
	xEP1908SenT_busy			: 		BOOL ;
	xEP1908SenT_Err				: 		BOOL ;
	udiEP1908SenT_ErrID			: 		UDINT ;

	// EP1908-002: 2-Channel Evaluation Error
	// The two channels contradict each other (not same value)
	fbEP1908_2CHEval_ADSRead	: 		ADSREAD ;
	wEP1908_2CHEval				: 		WORD ;
	xEP1908_2CHEval_busy		: 		BOOL ;
	xEP1908_2CHEval_Err			: 		BOOL ;
	udiEP1908_2CHEval_ErrID		: 		UDINT ;

	// EP1908-0002: Error In Safety Mat Operating Mode
	// Input pairs not in the same state (not same value)
	fbEP1908_SMiPair_ADSRead	: 		ADSREAD ;
	wEP1908_SMiPair				: 		WORD ;
	xEP1908_SMiPair_busy		: 		BOOL ;
	xEP1908_SMiPair_Err			: 		BOOL ;
	udiEP1908_SMiPair_ErrID		: 		UDINT ;

	// EP1908-0002: Error in Safety Mat Operating Supply
	// External supply detected (Input channel not getting test pulses)
	fbEP1908_SMExtSupply_ADSRead: ADSREAD;
	wEP1908_SMExtSupply			: 		WORD;
	xEP1908_SMExtSupply_busy	: 		BOOL;
	xEP1908_SMExtSupply_Err		: 		BOOL;
	udiEP1908_SMExtSupply_ErrID	: 		UDINT;

	// EP1908-0002: Error During Speed Monitoring
	// Frquency Greater Than 500Hz
	fbEP1908_FreqGT500_ADSRead	: 		ADSREAD ;
	wEP1908_FreqGT500			: 		WORD ;
	xEP1908_FreqGT500_busy		: 		BOOL ;
	xEP1908_FreqGT500_Err		: 		BOOL ;
	udiEP1908_FreqGT500_ErrID	: 		UDINT ;
	
	// EP1908-0002: Error In Operating Mode: Two Channel Sync Velocity Control
	// Both inputs of a "pair" cannot be inactive in this mode
	fbEP1908_BothInPairInact_ADSRead: ADSREAD ;
	wEP1908_BothInPairInact			: 	WORD ;
	xEP1908_BothInPairInact_busy	: 	BOOL ;
	xEP1908_BothInPairInact_Err		: 	BOOL ;
	udiEP1908_BothInPairInact_ErrID	: 	UDINT ;

	// EP1908-0002: Error In Operating Modes: Two Channel Sync Velocity Control and Two Channel Encoder Velocity Control
	// For a channel pair, two different motor speeds detected
	fbEP1908_PairUnequalFreq_ADSRead: 	ADSREAD ;
	wEP1908_PairUnequalFreq			: 	WORD ;
	xEP1908_PairUnequalFreq_busy	: 	BOOL ;
	xEP1908_PairUnequalFreq_Err		: 	BOOL ;
	udiEP1908_PairUnequalFreq_ErrID	: 	UDINT ;

	// EP1908-0002 FEATURES: Operating Mode
	fbEP1908_OperatingMode_ADSRead	: 	ADSREAD ;
	wEP1908_OperMode				: 	WORD ;
	xEP1908_OperMode_busy			: 	BOOL ;
	xEP1908_OperMode_Err			: 	BOOL ;
	udiEP1908_OperModeID			: 	UDINT ;

	//Sequence through 0x8001 FS Sensor Test
	iFS_Sensor_Test					: 	INT ;

	// EP1908-0002 FEATURES: Sensor Test Channel 1 Active/Inactive
	fbEP1908_STActive1_EcCoESdoRead	: 	FB_EcCoESdoRead ;
	bEP1908_STActive1				: 	BYTE ;
	xEP1908_STActive1_busy			: 	BOOL ;
	xEP1908_STActive1_Err			: 	BOOL ;
	udiEP1908_STActive1ID			: 	UDINT ;
	iCaseZeroScans					: 	INT ;
	
	// EP1908-0002 FEATURES: Sensor Test Channel 2 Active/Inactive
	fbEP1908_STActive2_EcCoESdoRead	: 	FB_EcCoESdoRead ;
	bEP1908_STActive2				: 	BYTE ;
	xEP1908_STActive2_busy			: 	BOOL ;
	xEP1908_STActive2_Err			: 	BOOL ;
	udiEP1908_STActive2ID			: 	UDINT ;
	iCaseOneScans					: 	INT ;
	
	// EP1908-0002 FEATURES: Sensor Test Channel 3 Active/Inactive
	fbEP1908_STActive3_EcCoESdoRead	: 	FB_EcCoESdoRead ;
	bEP1908_STActive3				: 	BYTE ;
	xEP1908_STActive3_busy			: 	BOOL ;
	xEP1908_STActive3_Err			: 	BOOL ;
	udiEP1908_STActive3ID			: 	UDINT ;
	iCaseTwoScans					: 	INT ;
	
	// EP1908-0002 FEATURES: Sensor Test Channel 4 Active/Inactive
	fbEP1908_STActive4_EcCoESdoRead	: 	FB_EcCoESdoRead ;
	bEP1908_STActive4				: 	BYTE ;
	xEP1908_STActive4_busy			: 	BOOL ;
	xEP1908_STActive4_Err			: 	BOOL ;
	udiEP1908_STActive4ID			: 	UDINT ;
	iCaseThreeScans					: 	INT ;
	
	// EP1908-0002 FEATURES: Sensor Test Channel 5 Active/Inactive
	fbEP1908_STActive5_EcCoESdoRead	: 	FB_EcCoESdoRead ;
	bEP1908_STActive5				: 	BYTE ;
	xEP1908_STActive5_busy			: 	BOOL ;
	xEP1908_STActive5_Err			: 	BOOL ;
	udiEP1908_STActive5ID			: 	UDINT ;
	iCaseFourScans					: 	INT ;
	
	// EP1908-0002 FEATURES: Sensor Test Channel 6 Active/Inactive
	fbEP1908_STActive6_EcCoESdoRead	: 	FB_EcCoESdoRead ;
	bEP1908_STActive6				: 	BYTE ;
	xEP1908_STActive6_busy			: 	BOOL ;
	xEP1908_STActive6_Err			: 	BOOL ;
	udiEP1908_STActive6ID			: 	UDINT ;
	iCaseFiveScans					: 	INT ;
	
	// EP1908-0002 FEATURES: Sensor Test Channel 7 Active/Inactive
	fbEP1908_STActive7_EcCoESdoRead	: 	FB_EcCoESdoRead ;
	bEP1908_STActive7				: 	BYTE ;
	xEP1908_STActive7_busy			: 	BOOL ;
	xEP1908_STActive7_Err			: 	BOOL ;
	udiEP1908_STActive7ID			: 	UDINT ;
	iCaseSixScans					: 	INT ;
	
	// EP1908-0002 FEATURES: Sensor Test Channel 8 Active/Inactive
	fbEP1908_STActive8_EcCoESdoRead	: 	FB_EcCoESdoRead ;
	bEP1908_STActive8				: 	BYTE ;
	xEP1908_STActive8_busy			: 	BOOL ;
	xEP1908_STActive8_Err			: 	BOOL ;
	udiEP1908_STActive8ID			: 	UDINT ;
	iCaseSevenScans					: 	INT ;

	//Sequence through 0x8002 FS Logic Of Input Pairs
	iFS_LogicOfInputPairs			: 	INT ;
	
	// EP1908-0002 FEATURES: Logic of Channels 1 and 2
	fbEP1908_Logic1_2_EcCoESdoRead	: 	FB_EcCoESdoRead ;
	bEP1908_Logic1_2				: 	BYTE ;
	xEP1908_Logic1_2_busy			: 	BOOL ;
	xEP1908_Logic1_2_Err			: 	BOOL ;
	udiEP1908_Logic1_2ID			: 	UDINT ;
	iCaseLogicZeroScans				: 	INT ;

	// EP1908-0002 FEATURES: Logic of Channels 3 and 4
	fbEP1908_Logic3_4_EcCoESdoRead	: 	FB_EcCoESdoRead ;
	bEP1908_Logic3_4				: 	BYTE ;
	xEP1908_Logic3_4_busy			: 	BOOL ;
	xEP1908_Logic3_4_Err			: 	BOOL ;
	udiEP1908_Logic3_4ID			: 	UDINT ;
	iCaseLogicOneScans				: 	INT ;
	
	// EP1908-0002 FEATURES: Logic of Channels 5 and 6
	fbEP1908_Logic5_6_EcCoESdoRead	: 	FB_EcCoESdoRead ;
	bEP1908_Logic5_6				: 	BYTE ;
	xEP1908_Logic5_6_busy			: 	BOOL ;
	xEP1908_Logic5_6_Err			: 	BOOL ;
	udiEP1908_Logic5_6ID			: 	UDINT ;
	iCaseLogicTwoScans				: 	INT ;
	
	// EP1908-0002 FEATURES: Logic of Channels 7 and 8
	fbEP1908_Logic7_8_EcCoESdoRead	: 	FB_EcCoESdoRead ;
	bEP1908_Logic7_8				: 	BYTE ;
	xEP1908_Logic7_8_busy			: 	BOOL ;
	xEP1908_Logic7_8_Err			: 	BOOL ;
	udiEP1908_Logic7_8ID			: 	UDINT ;
	iCaseLogicThreeScans			: 	INT ;

	//Sequence through 0x8003 FS Velocity Limits
	iFS_VelocityLimits				: 	INT ;
	
	// EP1908-0002 FEATURES: Velocity Limit Value Channel 1
	fbEP1908_VelLimit1_EcCoESdoRead	: 	FB_EcCoESdoRead ;
	wEP1908_VelLimit1				: 	WORD ;
	xEP1908_VelLimit1_busy			: 	BOOL ;
	xEP1908_VelLimit1_Err			: 	BOOL ;
	udiEP1908_VelLimit1ID			: 	UDINT ;
	iCaseVelLIMZeroScans			: 	INT ;
	
	// EP1908-0002 FEATURES: Velocity Limit Value Channel 2
	fbEP1908_VelLimit2_EcCoESdoRead	: 	FB_EcCoESdoRead ;
	wEP1908_VelLimit2				: 	WORD ;
	xEP1908_VelLimit2				: 	BOOL ;
	xEP1908_VelLimit2_busy			: 	BOOL ;
	xEP1908_VelLimit2_Err			: 	BOOL ;
	udiEP1908_VelLimit2ID			:	UDINT ;
	iCaseVelLIMOneScans				: 	INT ;

	// EP1908-0002 FEATURES: Velocity Limit Value Channel 3
	fbEP1908_VelLimit3_EcCoESdoRead	: 	FB_EcCoESdoRead ;
	wEP1908_VelLimit3				: 	WORD ;
	xEP1908_VelLimit3_busy			: 	BOOL ;
	xEP1908_VelLimit3_Err			: 	BOOL ;
	udiEP1908_VelLimit3ID			: 	UDINT ;
	iCaseVelLIMTwoScans				: 	INT ;
	
	// EP1908-0002 FEATURES: Velocity Limit Value Channel 4
	fbEP1908_VelLimit4_EcCoESdoRead	: 	FB_EcCoESdoRead ;
	wEP1908_VelLimit4				: 	WORD ;
	xEP1908_VelLimit4_busy			: 	BOOL ;
	xEP1908_VelLimit4_Err			: 	BOOL ;
	udiEP1908_VelLimit4ID			: 	UDINT ;
	iCaseVelLIMThreeScans			: 	INT ;
	
	// EP1908-0002 FEATURES: Velocity Limit Value Channel 5
	fbEP1908_VelLimit5_EcCoESdoRead	: 	FB_EcCoESdoRead ;
	wEP1908_VelLimit5				: 	WORD ;
	xEP1908_VelLimit5_busy			: 	BOOL ;
	xEP1908_VelLimit5_Err			:	BOOL ;
	udiEP1908_VelLimit5ID			: 	UDINT ;
	iCaseVelLIMFourScans			: 	INT ;
	
	// EP1908-0002 FEATURES: Velocity Limit Value Channel 6
	fbEP1908_VelLimit6_EcCoESdoRead	: 	FB_EcCoESdoRead ;
	wEP1908_VelLimit6				: 	WORD ;
	xEP1908_VelLimit6_busy			: 	BOOL ;
	xEP1908_VelLimit6_Err			: 	BOOL ;
	udiEP1908_VelLimit6ID			: 	UDINT ;
	iCaseVelLIMFiveScans				: 	INT ;
	
	// EP1908-0002 FEATURES: Velocity Limit Value Channel 7
	fbEP1908_VelLimit7_EcCoESdoRead	: 	FB_EcCoESdoRead ;
	wEP1908_VelLimit7				: 	WORD ;
	xEP1908_VelLimit7_busy			: 	BOOL ;
	xEP1908_VelLimit7_Err			: 	BOOL ;
	udiEP1908_VelLimit7ID			: 	UDINT ;
	iCaseVelLIMSixScans				: 	INT ;
	
	// EP1908-0002 FEATURES: Velocity Limit Value Channel 8
	fbEP1908_VelLimit8_EcCoESdoRead	: 	FB_EcCoESdoRead ;
	wEP1908_VelLimit8				: 	WORD ;
	xEP1908_VelLimit8_busy			: 	BOOL ;
	xEP1908_VelLimit8_Err			: 	BOOL ; 
	udiEP1908_VelLimit8ID			: 	UDINT ;
	iCaseVelLIMSevenScans			: 	INT ;
END_VAR
VAR_INPUT
END_VAR

//		8-2-2012
// 		This Program has been supplied by Beckhoff Automation As-Is and is intended only as an example 
//		implementation. Functionality is not guaranteed. 
//
IF g_bHMI_ScreenBeingDisplayed = 20 THEN
// Interval timer for CoE Reads
T1(
						IN				:= 		NOT xExecute, 
						PT				:=		T#500MS, 
						Q				=>		xExecute, 
						ET				=>		tTime1 ) ;

C1(
						CU				:= 		xExecute, 
						RESET			:= 		xReset, 
						PV				:= 		wPreset, 
						Q				=> 		xDone, 
						CV				=> 		wCount) ;

IF C1.CV > 8 	THEN xReset := 1 ;
				ELSE xReset := 0 ; 
END_IF ;

// Read the serial number out of the EP1908-0002
fbEP1908Sn_ADSRead(
						NETID			:= 		gc_sADSNetID, 
						PORT			:= 		gc_uiEP1908_EtherCATAdr, 
						IDXGRP			:= 		16#F302, 
						IDXOFFS			:= 		16#F9800002, 
						LEN				:= 		4, 
						DESTADDR		:= 		ADR(dwEP1908_Sn), 
						READ			:= 		xExecute, 
						TMOUT			:= 		T#2S, 
						BUSY			=> 		xEP1908Sn_busy, 
						ERR				=> 		xEP1908Sn_Err, 
						ERRID			=> 		xEP1908Sn_ErrID );

g_dwHMI_EP1908Sn 						:= 		dwEP1908_Sn ;

// Read the DIP Switch Setting out of the EP1908-0002
IF C1.CV = 1 THEN
fbEP1908DSw_ADSRead(
						NETID			:= 		gc_sADSNetID, 
						PORT			:= 		gc_uiEP1908_EtherCATAdr, 
						IDXGRP			:= 		16#F302, 
						IDXOFFS			:= 		16#F9800001, 
						LEN				:= 		2, 
						DESTADDR		:= 		ADR(wEP1908_DSw), 
						READ			:= 		xExecute, 
						TMOUT			:= 		T#2S, 
						BUSY			=> 		xEP1908DSw_busy, 
						ERR				=> 		xEP1908DSw_Err, 
						ERRID			=> 		udiEP1908DSw_ErrID );

g_wHMI_EP1908DSw 						:= 		wEP1908_DSw ;
END_IF ;						

//Read the Hardware Version of the EP1908-0002 Terminal
fbEP1908_HWvers_EcCoESdoRead(
						sNetId			:= 		gc_sADSNetID, 
						nSlaveAddr		:= 		gc_uiEP1908_EtherCATAdr, 
						nSubIndex		:= 		0, 
						nIndex			:= 		16#1009, 
						pDstBuf			:=  	ADR(sEP1908_HWvers),
						cbBufLen		:= 		SIZEOF(sEP1908_HWvers), 
						bExecute		:= 		xExecute, 
						tTimeout		:= 		T#2S, 
						bBusy			=> 		xEP1908_HWvers_Busy, 
						bError			=> 		xEP1908_HWvers_Err, 
						nErrId			=> 		udiEP1908_HWvers_ErrID ) ;

g_sHMI_EP1908_HWvers					:= 		sEP1908_HWvers ;

//Read the Software Version of the EP1908-002 Logic Terminal (It's f/w)
fbEP1908_FWvers_EcCoESdoRead(
						sNetId			:= 		gc_sADSNetID, 
						nSlaveAddr		:= 		gc_uiEP1908_EtherCATAdr, 
						nSubIndex		:= 		0, 
						nIndex			:= 		16#100A, 
						pDstBuf			:=  	ADR(sEP1908_FWvers),
						cbBufLen		:= 		SIZEOF(sEP1908_FWvers), 
						bExecute		:= 		xExecute, 
						tTimeout		:= 		T#2S, 
						bBusy			=> 		xEP1908_FWvers_Busy, 
						bError			=> 		xEP1908_FWvers_Err, 
						nErrId			=> 		udiEP1908_FWvers_ErrID ) ;
						
g_sHMI_EP1908_FWvers					:= 		sEP1908_FWvers ;

// EP1908-0002 FEATURES: Operating Mode
fbEP1908_OperatingMode_ADSRead(
						NETID			:= 		gc_sADSNetID, 
						PORT			:= 		gc_uiEP1908_EtherCATAdr, 
						IDXGRP			:= 		16#F302, 
						IDXOFFS			:= 		16#80000001, 
						LEN				:= 		2, 
						DESTADDR		:=		ADR(wEP1908_OperMode), 
						READ			:= 		xExecute, 
						TMOUT			:= 		T#2S, 
						BUSY			=> 		xEP1908_OperMode_busy, 
						ERR				=> 		xEP1908_OperMode_Err, 
						ERRID			=> 		udiEP1908_OperModeID );
		
IF wEP1908_OperMode 					= 		0 THEN
	g_sHMI_EP1908_OperatingMode 		:= 		'Digital' ;
	ELSIF wEP1908_OperMode 				= 		1 THEN
	g_sHMI_EP1908_OperatingMode 		:= 		'Standstill Monitoring 1' ;
	ELSIF wEP1908_OperMode 				= 		2 THEN
	g_sHMI_EP1908_OperatingMode 		:= 		'Standstill Monitoring 2' ;
ELSE
	g_sHMI_EP1908_OperatingMode 		:= 		'Invalid Mode' ;
END_IF ;


CASE iFS_Sensor_Test OF

0:
// EP1908-0002 FEATURES: Sensor Test Channel 1 Active/Inactive
iCaseSevenScans 						:= 		0 ;
fbEP1908_STActive1_EcCoESdoRead(
						sNetId			:= 		gc_sADSNetID, 
						nSlaveAddr		:= 		gc_uiEP1908_EtherCATAdr, 
						nSubIndex		:= 		1, 
						nIndex			:= 		16#8001, 
						pDstBuf			:= 		ADR(bEP1908_STActive1), 
						cbBufLen		:= 		SIZEOF(bEP1908_STActive1), 
						bExecute		:= 		xExecute, 
						tTimeout		:= 		T#2S, 
						bBusy			=> 		xEP1908_STActive1_busy, 
						bError			=> 		xEP1908_STActive1_Err, 
						nErrId			=> 		udiEP1908_STActive1ID );

g_xHMI_EP1908_SensTestActive1			:= 		bEP1908_STActive1.0 ;

iCaseZeroScans := iCaseZeroScans + 1 ; //Prevent code from passing through in only one pass

IF NOT xEP1908_STActive1_busy AND NOT xEP1908_STActive1_Err AND iCaseZeroScans <> 0 THEN
	iFS_Sensor_Test := 1 ;
END_IF ;

1:
// EP1908-0002 FEATURES: Sensor Test Channel 2 Active/Inactive
iCaseZeroScans 							:= 		0 ;
fbEP1908_STActive2_EcCoESdoRead(
						sNetId			:= 		gc_sADSNetID, 
						nSlaveAddr		:= 		gc_uiEP1908_EtherCATAdr, 
						nSubIndex		:= 		2, 
						nIndex			:= 		16#8001, 
						pDstBuf			:= 		ADR(bEP1908_STActive2), 
						cbBufLen		:= 		SIZEOF(bEP1908_STActive2), 
						bExecute		:= 		xExecute, 
						tTimeout		:= 		T#2S, 
						bBusy			=> 		xEP1908_STActive2_busy, 
						bError			=> 		xEP1908_STActive2_Err, 
						nErrId			=> 		udiEP1908_STActive2ID );

g_xHMI_EP1908_SensTestActive2			:= 		bEP1908_STActive2.0 ;

iCaseOneScans := iCaseOneScans + 1 ; //Prevent code from passing through in only one pass

IF NOT xEP1908_STActive2_busy AND NOT xEP1908_STActive2_Err AND iCaseOneScans <> 0 THEN
	iFS_Sensor_Test := 2 ;
END_IF ;

2:
// EP1908-0002 FEATURES: Sensor Test Channel 3 Active/Inactive
iCaseOneScans := 0 ;
fbEP1908_STActive3_EcCoESdoRead(
						sNetId			:= 		gc_sADSNetID, 
						nSlaveAddr		:= 		gc_uiEP1908_EtherCATAdr, 
						nSubIndex		:= 		3, 
						nIndex			:= 		16#8001, 
						pDstBuf			:= 		ADR(bEP1908_STActive3), 
						cbBufLen		:= 		SIZEOF(bEP1908_STActive3), 
						bExecute		:= 		xExecute, 
						tTimeout		:= 		T#2S, 
						bBusy			=> 		xEP1908_STActive3_busy, 
						bError			=> 		xEP1908_STActive3_Err, 
						nErrId			=> 		udiEP1908_STActive3ID );

g_xHMI_EP1908_SensTestActive3			:= 		bEP1908_STActive3.0 ;

iCaseTwoScans := iCaseTwoScans + 1 ; //Prevent code from passing through in only one pass

IF NOT xEP1908_STActive3_busy AND NOT xEP1908_STActive3_Err AND iCaseTwoScans <> 0 THEN
	iFS_Sensor_Test := 3 ;
END_IF ;

3:
// EP1908-0002 FEATURES: Sensor Test Channel 4 Active/Inactive
iCaseTwoScans := 0 ;
fbEP1908_STActive4_EcCoESdoRead(
						sNetId			:= 		gc_sADSNetID, 
						nSlaveAddr		:= 		gc_uiEP1908_EtherCATAdr, 
						nSubIndex		:= 		4, 
						nIndex			:= 		16#8001, 
						pDstBuf			:= 		ADR(bEP1908_STActive4), 
						cbBufLen		:= 		SIZEOF(bEP1908_STActive4), 
						bExecute		:= 		xExecute, 
						tTimeout		:= 		T#2S, 
						bBusy			=> 		xEP1908_STActive4_busy, 
						bError			=> 		xEP1908_STActive4_Err, 
						nErrId			=> 		udiEP1908_STActive4ID );

g_xHMI_EP1908_SensTestActive4			:= 		bEP1908_STActive4.0 ;

iCaseThreeScans := iCaseThreeScans + 1 ; //Prevent code from passing through in only one pass

IF NOT xEP1908_STActive4_busy AND NOT xEP1908_STActive4_Err AND iCaseThreeScans <> 0 THEN
	iFS_Sensor_Test := 4 ;
END_IF ;

4:
// EP1908-0002 FEATURES: Sensor Test Channel 5 Active/Inactive
iCaseThreeScans := 0 ;
fbEP1908_STActive5_EcCoESdoRead(
						sNetId			:= 		gc_sADSNetID, 
						nSlaveAddr		:= 		gc_uiEP1908_EtherCATAdr, 
						nSubIndex		:= 		5, 
						nIndex			:= 		16#8001, 
						pDstBuf			:= 		ADR(bEP1908_STActive5), 
						cbBufLen		:= 		SIZEOF(bEP1908_STActive5), 
						bExecute		:= 		xExecute, 
						tTimeout		:= 		T#2S, 
						bBusy			=> 		xEP1908_STActive5_busy, 
						bError			=> 		xEP1908_STActive5_Err, 
						nErrId			=> 		udiEP1908_STActive5ID );

g_xHMI_EP1908_SensTestActive5			:= 		bEP1908_STActive5.0 ;

iCaseFourScans := iCaseFourScans + 1 ; //Prevent code from passing through in only one pass

IF NOT xEP1908_STActive5_busy AND NOT xEP1908_STActive5_Err AND iCaseFourScans <> 0 THEN
	iFS_Sensor_Test := 5 ;
END_IF ;

5:
// EP1908-0002 FEATURES: Sensor Test Channel 6 Active/Inactive
iCaseFourScans := 0 ;
fbEP1908_STActive6_EcCoESdoRead(
						sNetId			:= 		gc_sADSNetID, 
						nSlaveAddr		:= 		gc_uiEP1908_EtherCATAdr, 
						nSubIndex		:= 		6, 
						nIndex			:= 		16#8001, 
						pDstBuf			:= 		ADR(bEP1908_STActive6), 
						cbBufLen		:= 		SIZEOF(bEP1908_STActive6), 
						bExecute		:= 		xExecute, 
						tTimeout		:= 		T#2S, 
						bBusy			=> 		xEP1908_STActive6_busy, 
						bError			=> 		xEP1908_STActive6_Err, 
						nErrId			=> 		udiEP1908_STActive6ID );

g_xHMI_EP1908_SensTestActive6			:= 		bEP1908_STActive6.0 ;

iCaseFiveScans := iCaseFiveScans + 1 ; //Prevent code from passing through in only one pass

IF NOT xEP1908_STActive6_busy AND NOT xEP1908_STActive6_Err AND iCaseFiveScans <> 0 THEN
	iFS_Sensor_Test := 6 ;
END_IF ;

6:
// EP1908-0002 FEATURES: Sensor Test Channel 7 Active/Inactive
iCaseFiveScans := 0 ;
fbEP1908_STActive7_EcCoESdoRead(
						sNetId			:= 		gc_sADSNetID, 
						nSlaveAddr		:= 		gc_uiEP1908_EtherCATAdr, 
						nSubIndex		:= 		7, 
						nIndex			:= 		16#8001, 
						pDstBuf			:= 		ADR(bEP1908_STActive7), 
						cbBufLen		:= 		SIZEOF(bEP1908_STActive7), 
						bExecute		:= 		xExecute, 
						tTimeout		:= 		T#2S, 
						bBusy			=> 		xEP1908_STActive7_busy, 
						bError			=> 		xEP1908_STActive7_Err, 
						nErrId			=> 		udiEP1908_STActive7ID );

g_xHMI_EP1908_SensTestActive7			:= 		bEP1908_STActive7.0 ;

iCaseSixScans := iCaseSixScans + 1 ; //Prevent code from passing through in only one pass

IF NOT xEP1908_STActive7_busy AND NOT xEP1908_STActive7_Err AND iCaseSixScans <> 0 THEN
	iFS_Sensor_Test := 7 ;
END_IF ;

7:
// EP1908-0002 FEATURES: Sensor Test Channel 8 Active/Inactive
iCaseSixScans := 0 ;
fbEP1908_STActive8_EcCoESdoRead(
						sNetId			:= 		gc_sADSNetID, 
						nSlaveAddr		:= 		gc_uiEP1908_EtherCATAdr, 
						nSubIndex		:= 		8, 
						nIndex			:= 		16#8001, 
						pDstBuf			:= 		ADR(bEP1908_STActive8), 
						cbBufLen		:= 		SIZEOF(bEP1908_STActive8), 
						bExecute		:= 		xExecute, 
						tTimeout		:= 		T#2S, 
						bBusy			=> 		xEP1908_STActive8_busy, 
						bError			=> 		xEP1908_STActive8_Err, 
						nErrId			=> 		udiEP1908_STActive8ID );

g_xHMI_EP1908_SensTestActive8			:= 		bEP1908_STActive8.0 ;

iCaseSevenScans := iCaseSevenScans + 1 ; //Prevent code from passing through in only one pass

IF NOT xEP1908_STActive8_busy AND NOT xEP1908_STActive8_Err AND iCaseSevenScans <> 0 THEN
	iFS_Sensor_Test := 0 ;
END_IF ;
	END_CASE ;


//Sequence through 0x8002 FS Logic Of Input Pairs
CASE iFS_LogicOfInputPairs OF

0:
// EP1908-0002 FEATURES: Logic of Channels 1 and 2
iCaseLogicThreeScans 					:= 		0 ;
fbEP1908_Logic1_2_EcCoESdoRead(
						sNetId			:= 		gc_sADSNetID, 
						nSlaveAddr		:= 		gc_uiEP1908_EtherCATAdr, 
						nSubIndex		:= 		1, 
						nIndex			:= 		16#8002, 
						pDstBuf			:= 		ADR(bEP1908_Logic1_2), 
						cbBufLen		:= 		SIZEOF(bEP1908_Logic1_2), 
						bExecute		:= 		xExecute, 
						tTimeout		:= 		T#2S, 
						bBusy			=> 		xEP1908_Logic1_2_busy, 
						bError			=> 		xEP1908_Logic1_2_Err, 
						nErrId			=> 		udiEP1908_Logic1_2ID );

IF bEP1908_Logic1_2 					= 		0 THEN
	g_sHMI_EP1908_LogicCh1andCh2 		:= 		'Single Channel Logic' ;
	ELSIF bEP1908_Logic1_2 				= 		1 THEN
	g_sHMI_EP1908_LogicCh1andCh2 		:= 		'Asynchronous Analysis OSSD, Sensor Test Must Be Disabled!' ;
	ELSIF bEP1908_Logic1_2 				= 		2 THEN
	g_sHMI_EP1908_LogicCh1andCh2 		:= 		'Any Pulse Repetitive OSSD, Sensor Test Must Be Disabled!' ;
	ELSIF bEP1908_Logic1_2 				= 		3 THEN
	g_sHMI_EP1908_LogicCh1andCh2 		:= 		'Short Cut, No Module Fault (Safety Mat Operation)' ;
	ELSIF bEP1908_Logic1_2 				= 		4 THEN
	g_sHMI_EP1908_LogicCh1andCh2 		:= 		'Velocity Control Ch1 / Single Channel Logic Ch2' ;
	ELSIF bEP1908_Logic1_2 				= 		5 THEN
	g_sHMI_EP1908_LogicCh1andCh2 		:= 		'Single Channel Logic Ch1 / Velocity Control Ch2' ;
	ELSIF bEP1908_Logic1_2 				= 		6 THEN
	g_sHMI_EP1908_LogicCh1andCh2 		:= 		'Velocity Control For Both Ch1 and Ch2' ;
	ELSIF bEP1908_Logic1_2 				= 		7 THEN
	g_sHMI_EP1908_LogicCh1andCh2 		:= 		'Two Channel Sync Velocity (Speed Monitoring Prox.es)' ;
	ELSIF bEP1908_Logic1_2 				= 		8 THEN
	g_sHMI_EP1908_LogicCh1andCh2 		:= 		'Two Channel Encoder Velocity (Speed Monitoring Encoder)' ;
	ELSIF bEP1908_Logic1_2 				= 		9 THEN
	g_sHMI_EP1908_LogicCh1andCh2 		:= 		'Two Channel Asynch Velocity (Prox Switches)' ;	
ELSE
	g_sHMI_EP1908_LogicCh1andCh2 		:= 		'Invalid Logic CH1 and CH2' ;
END_IF ;						

iCaseLogicZeroScans := iCaseLogicZeroScans + 1 ; //Prevent code from passing through in only one pass

IF NOT xEP1908_Logic1_2_busy AND NOT xEP1908_Logic1_2_Err AND iCaseLogicZeroScans <> 0 THEN
	iFS_LogicOfInputPairs := 1 ;
END_IF ;

1:			
// EP1908-0002 FEATURES: Logic of Channels 3 and 4
iCaseLogicZeroScans := 0 ;
fbEP1908_Logic3_4_EcCoESdoRead(
						sNetId			:= 		gc_sADSNetID, 
						nSlaveAddr		:= 		gc_uiEP1908_EtherCATAdr, 
						nSubIndex		:= 		5, 
						nIndex			:= 		16#8002, 
						pDstBuf			:= 		ADR(bEP1908_Logic3_4), 
						cbBufLen		:= 		SIZEOF(bEP1908_Logic3_4), 
						bExecute		:= 		xExecute, 
						tTimeout		:= 		T#2S, 
						bBusy			=> 		xEP1908_Logic3_4_busy, 
						bError			=> 		xEP1908_Logic3_4_Err, 
						nErrId			=> 		udiEP1908_Logic3_4ID );

IF bEP1908_Logic3_4 					= 		0 THEN
	g_sHMI_EP1908_LogicCh3andCh4 		:= 		'Single Channel Logic' ;
	ELSIF bEP1908_Logic3_4 				= 		1 THEN
	g_sHMI_EP1908_LogicCh3andCh4 		:= 		'Asynchronous Analysis OSSD, Sensor Test Must Be Disabled!' ;
	ELSIF bEP1908_Logic3_4 				= 		2 THEN
	g_sHMI_EP1908_LogicCh3andCh4 		:= 		'Any Pulse Repetitive OSSD, Sensor Test Must Be Disabled!' ;
	ELSIF bEP1908_Logic3_4 				= 		3 THEN
	g_sHMI_EP1908_LogicCh3andCh4 		:= 		'Short Cut, No Module Fault (Safety Mat Operation)' ;
	ELSIF bEP1908_Logic3_4 				= 		4 THEN
	g_sHMI_EP1908_LogicCh3andCh4 		:= 		'Velocity Control Ch3 / Single Channel Logic Ch4' ;
	ELSIF bEP1908_Logic3_4 				= 		5 THEN
	g_sHMI_EP1908_LogicCh3andCh4 		:= 		'Single Channel Logic Ch3 / Velocity Control Ch4' ;
	ELSIF bEP1908_Logic3_4 				= 		6 THEN
	g_sHMI_EP1908_LogicCh3andCh4 		:= 		'Velocity Control For Both Ch3 and Ch4' ;
	ELSIF bEP1908_Logic3_4 				= 		7 THEN
	g_sHMI_EP1908_LogicCh3andCh4 		:= 		'Two Channel Sync Velocity (Speed Monitoring Prox.es)' ;
	ELSIF bEP1908_Logic3_4 				= 		8 THEN
	g_sHMI_EP1908_LogicCh3andCh4 		:= 		'Two Channel Encoder Velocity (Speed Monitoring Encoder)' ;
	ELSIF bEP1908_Logic3_4 				= 		9 THEN
	g_sHMI_EP1908_LogicCh3andCh4 		:= 		'Two Channel Asynch Velocity (Prox Switches)' ;	
ELSE
	g_sHMI_EP1908_LogicCh3andCh4 		:= 		'Invalid Logic CH3 and CH4' ;
END_IF ;						

iCaseLogicOneScans := iCaseLogicOneScans + 1 ; //Prevent code from passing through in only one pass

IF NOT xEP1908_Logic3_4_busy AND NOT xEP1908_Logic3_4_Err AND iCaseLogicOneScans <> 0 THEN
	iFS_LogicOfInputPairs := 2 ;
END_IF ;
	
2:
// EP1908-0002 FEATURES: Logic of Channels 5 and 6
iCaseLogicOneScans := 0 ;
fbEP1908_Logic5_6_EcCoESdoRead(
						sNetId			:= 		gc_sADSNetID, 
						nSlaveAddr		:= 		gc_uiEP1908_EtherCATAdr, 
						nSubIndex		:= 		9, 
						nIndex			:= 		16#8002, 
						pDstBuf			:= 		ADR(bEP1908_Logic5_6), 
						cbBufLen		:= 		SIZEOF(bEP1908_Logic5_6), 
						bExecute		:= 		xExecute, 
						tTimeout		:= 		T#2S, 
						bBusy			=> 		xEP1908_Logic5_6_busy, 
						bError			=> 		xEP1908_Logic5_6_Err, 
						nErrId			=> 		udiEP1908_Logic5_6ID );

IF bEP1908_Logic5_6 					= 		0 THEN
	g_sHMI_EP1908_LogicCh5andCh6 		:= 		'Single Channel Logic' ;
	ELSIF bEP1908_Logic5_6 				= 		1 THEN
	g_sHMI_EP1908_LogicCh5andCh6 		:= 		'Asynchronous Analysis OSSD, Sensor Test Must Be Disabled!' ;
	ELSIF bEP1908_Logic5_6 				= 		2 THEN
	g_sHMI_EP1908_LogicCh5andCh6 		:= 		'Any Pulse Repetitive OSSD, Sensor Test Must Be Disabled!' ;
	ELSIF bEP1908_Logic5_6 				= 		3 THEN
	g_sHMI_EP1908_LogicCh5andCh6 		:= 		'Short Cut, No Module Fault (Safety Mat Operation)' ;
	ELSIF bEP1908_Logic5_6 				= 		4 THEN
	g_sHMI_EP1908_LogicCh5andCh6 		:= 		'Velocity Control Ch5 / Single Channel Logic Ch6' ;
	ELSIF bEP1908_Logic5_6 				= 		5 THEN
	g_sHMI_EP1908_LogicCh5andCh6 		:= 		'Single Channel Logic Ch5 / Velocity Control Ch6' ;
	ELSIF bEP1908_Logic5_6 				= 		6 THEN
	g_sHMI_EP1908_LogicCh5andCh6 		:= 		'Velocity Control For Both Ch5 and Ch6' ;
	ELSIF bEP1908_Logic5_6 				= 		7 THEN
	g_sHMI_EP1908_LogicCh5andCh6 		:= 		'Two Channel Sync Velocity (Speed Monitoring Prox.es)' ;
	ELSIF bEP1908_Logic5_6 				= 		8 THEN
	g_sHMI_EP1908_LogicCh5andCh6 		:= 		'Two Channel Encoder Velocity (Speed Monitoring Encoder)' ;
	ELSIF bEP1908_Logic5_6 				= 		9 THEN
	g_sHMI_EP1908_LogicCh5andCh6 		:= 		'Two Channel Asynch Velocity (Prox Switches)' ;	
ELSE
	g_sHMI_EP1908_LogicCh5andCh6 		:= 		'Invalid Logic CH5 and CH6' ;
END_IF ;		

iCaseLogicTwoScans := iCaseLogicTwoScans + 1 ; //Prevent code from passing through in only one pass

IF NOT xEP1908_Logic5_6_busy AND NOT xEP1908_Logic5_6_Err AND iCaseLogicTwoScans <> 0 THEN
	iFS_LogicOfInputPairs := 3 ;
END_IF ;

3:
// EP1908-0002 FEATURES: Logic of Channels 7 and 8
iCaseLogicTwoScans := 0 ;
fbEP1908_Logic7_8_EcCoESdoRead(
						sNetId			:= 		gc_sADSNetID, 
						nSlaveAddr		:= 		gc_uiEP1908_EtherCATAdr, 
						nSubIndex		:= 		16#D, 
						nIndex			:= 		16#8002, 
						pDstBuf			:= 		ADR(bEP1908_Logic7_8), 
						cbBufLen		:= 		SIZEOF(bEP1908_Logic7_8), 
						bExecute		:= 		xExecute, 
						tTimeout		:= 		T#2S, 
						bBusy			=> 		xEP1908_Logic7_8_busy, 
						bError			=> 		xEP1908_Logic7_8_Err, 
						nErrId			=> 		udiEP1908_Logic7_8ID );

IF bEP1908_Logic7_8 					= 		0 THEN
	g_sHMI_EP1908_LogicCh7andCh8 		:= 		'Single Channel Logic' ;
	ELSIF bEP1908_Logic7_8 				= 		1 THEN
	g_sHMI_EP1908_LogicCh7andCh8 		:= 		'Asynchronous Analysis OSSD, Sensor Test Must Be Disabled!' ;
	ELSIF bEP1908_Logic7_8 				= 		2 THEN
	g_sHMI_EP1908_LogicCh7andCh8 		:= 		'Any Pulse Repetitive OSSD, Sensor Test Must Be Disabled!' ;
	ELSIF bEP1908_Logic7_8 				= 		3 THEN
	g_sHMI_EP1908_LogicCh7andCh8 		:= 		'Short Cut, No Module Fault (Safety Mat Operation)' ;
	ELSIF bEP1908_Logic7_8 				= 		4 THEN
	g_sHMI_EP1908_LogicCh7andCh8 		:= 		'Velocity Control Ch7 / Single Channel Logic Ch8' ;
	ELSIF bEP1908_Logic7_8 				= 		5 THEN
	g_sHMI_EP1908_LogicCh7andCh8 		:= 		'Single Channel Logic Ch7 / Velocity Control Ch8' ;
	ELSIF bEP1908_Logic7_8 				= 		6 THEN
	g_sHMI_EP1908_LogicCh7andCh8 		:= 		'Velocity Control For Both Ch7 and Ch8' ;
	ELSIF bEP1908_Logic7_8 				= 		7 THEN
	g_sHMI_EP1908_LogicCh7andCh8 		:= 		'Two Channel Sync Velocity (Speed Monitoring Prox.es)' ;
	ELSIF bEP1908_Logic7_8 				= 		8 THEN
	g_sHMI_EP1908_LogicCh7andCh8 		:= 		'Two Channel Encoder Velocity (Speed Monitoring Encoder)' ;
	ELSIF bEP1908_Logic7_8 				= 		9 THEN
	g_sHMI_EP1908_LogicCh7andCh8 		:= 		'Two Channel Asynch Velocity (Prox Switches)' ;	
ELSE
	g_sHMI_EP1908_LogicCh7andCh8 		:= 		'Invalid Logic CH7 and CH8' ;
END_IF ;

iCaseLogicThreeScans := iCaseLogicThreeScans + 1 ; //Prevent code from passing through in only one pass

IF NOT xEP1908_Logic7_8_busy AND NOT xEP1908_Logic7_8_Err AND iCaseLogicThreeScans <> 0 THEN
	iFS_LogicOfInputPairs := 0 ;
END_IF ;
END_CASE ;


CASE iFS_VelocityLimits OF

0:
// EP1908-0002 FEATURES: Velocity Limit Channel 1
iCaseVelLIMSevenScans := 0 ;
fbEP1908_VelLimit1_EcCoESdoRead(
						sNetId			:= 		gc_sADSNetID, 
						nSlaveAddr		:= 		gc_uiEP1908_EtherCATAdr, 
						nSubIndex		:= 		1, 
						nIndex			:= 		16#8003, 
						pDstBuf			:= 		ADR(wEP1908_VelLimit1), 
						cbBufLen		:= 		SIZEOF(wEP1908_VelLimit1), 
						bExecute		:= 		xExecute, 
						tTimeout		:= 		T#2S, 
						bBusy			=> 		xEP1908_VelLimit1_busy, 
						bError			=> 		xEP1908_VelLimit1_Err, 
						nErrId			=> 		udiEP1908_VelLimit1ID );

g_wHMI_EP1908_VelLimit1					:= 		wEP1908_VelLimit1 ;

iCaseVelLIMZeroScans := iCaseVelLIMZeroScans + 1 ; //Prevent code from passing through in only one pass

IF NOT xEP1908_VelLimit1_busy AND NOT xEP1908_VelLimit1_Err AND iCaseVelLIMZeroScans <> 0 THEN
	iFS_VelocityLimits := 1 ;
END_IF ;

1:
// EP1908-0002 FEATURES: Velocity Limit Channel 2
iCaseVelLIMZeroScans := 0 ;
fbEP1908_VelLimit2_EcCoESdoRead(
						sNetId			:= 		gc_sADSNetID, 
						nSlaveAddr		:= 		gc_uiEP1908_EtherCATAdr, 
						nSubIndex		:= 		2, 
						nIndex			:= 		16#8003, 
						pDstBuf			:= 		ADR(wEP1908_VelLimit2), 
						cbBufLen		:= 		SIZEOF(wEP1908_VelLimit2), 
						bExecute		:= 		xExecute, 
						tTimeout		:= 		T#2S, 
						bBusy			=> 		xEP1908_VelLimit2_busy, 
						bError			=> 		xEP1908_VelLimit2_Err, 
						nErrId			=> 		udiEP1908_VelLimit2ID );

g_wHMI_EP1908_VelLimit2					:= 		wEP1908_VelLimit2 ;

iCaseVelLIMOneScans := iCaseVelLIMOneScans + 1 ; //Prevent code from passing through in only one pass

IF NOT xEP1908_VelLimit2_busy AND NOT xEP1908_VelLimit2_Err AND iCaseVelLIMOneScans <> 0 THEN
	iFS_VelocityLimits := 2 ;
END_IF ;

2:
// EP1908-0002 FEATURES: Velocity Limit Channel 3
iCaseVelLIMOneScans := 0 ;
fbEP1908_VelLimit3_EcCoESdoRead(
						sNetId			:= 		gc_sADSNetID, 
						nSlaveAddr		:= 		gc_uiEP1908_EtherCATAdr, 
						nSubIndex		:= 		3, 
						nIndex			:= 		16#8003, 
						pDstBuf			:= 		ADR(wEP1908_VelLimit3), 
						cbBufLen		:= 		SIZEOF(wEP1908_VelLimit3), 
						bExecute		:= 		xExecute, 
						tTimeout		:= 		T#2S, 
						bBusy			=> 		xEP1908_VelLimit3_busy, 
						bError			=> 		xEP1908_VelLimit3_Err, 
						nErrId			=> 		udiEP1908_VelLimit3ID );

g_wHMI_EP1908_VelLimit3					:= 		wEP1908_VelLimit3 ;

iCaseVelLIMTwoScans := iCaseVelLIMTwoScans + 1 ; //Prevent code from passing through in only one pass

IF NOT xEP1908_VelLimit3_busy AND NOT xEP1908_VelLimit3_Err AND iCaseVelLIMTwoScans <> 0 THEN
	iFS_VelocityLimits := 3 ;
END_IF ;

3:
// EP1908-0002 FEATURES: Velocity Limit Channel 4
iCaseVelLIMTwoScans := 0 ;
fbEP1908_VelLimit4_EcCoESdoRead(
						sNetId			:= 		gc_sADSNetID, 
						nSlaveAddr		:= 		gc_uiEP1908_EtherCATAdr, 
						nSubIndex		:= 		4, 
						nIndex			:= 		16#8003, 
						pDstBuf			:= 		ADR(wEP1908_VelLimit4), 
						cbBufLen		:= 		SIZEOF(wEP1908_VelLimit4), 
						bExecute		:= 		xExecute, 
						tTimeout		:= 		T#2S, 
						bBusy			=> 		xEP1908_VelLimit4_busy, 
						bError			=> 		xEP1908_VelLimit4_Err, 
						nErrId			=> 		udiEP1908_VelLimit4ID );

g_wHMI_EP1908_VelLimit4					:= 		wEP1908_VelLimit4 ;

iCaseVelLIMThreeScans := iCaseVelLIMThreeScans + 1 ; //Prevent code from passing through in only one pass

IF NOT xEP1908_VelLimit4_busy AND NOT xEP1908_VelLimit4_Err AND iCaseVelLIMThreeScans <> 0 THEN
	iFS_VelocityLimits := 4 ;
END_IF ;

4:
// EP1908-0002 FEATURES: Velocity Limit Channel 5
iCaseVelLIMThreeScans := 0 ;
fbEP1908_VelLimit5_EcCoESdoRead(
						sNetId			:= 		gc_sADSNetID, 
						nSlaveAddr		:= 		gc_uiEP1908_EtherCATAdr, 
						nSubIndex		:= 		5, 
						nIndex			:= 		16#8003, 
						pDstBuf			:= 		ADR(wEP1908_VelLimit5), 
						cbBufLen		:= 		SIZEOF(wEP1908_VelLimit5), 
						bExecute		:= 		xExecute, 
						tTimeout		:= 		T#2S, 
						bBusy			=> 		xEP1908_VelLimit5_busy, 
						bError			=> 		xEP1908_VelLimit5_Err, 
						nErrId			=> 		udiEP1908_VelLimit5ID );

g_wHMI_EP1908_VelLimit5					:= 		wEP1908_VelLimit5 ;

iCaseVelLIMFourScans := iCaseVelLIMFourScans + 1 ; //Prevent code from passing through in only one pass

IF NOT xEP1908_VelLimit5_busy AND NOT xEP1908_VelLimit5_Err AND iCaseVelLIMFourScans <> 0 THEN
	iFS_VelocityLimits := 5 ;
END_IF ;

5:
// EP1908-0002 FEATURES: Velocity Limit Channel 6
iCaseVelLIMFourScans := 0 ;
fbEP1908_VelLimit6_EcCoESdoRead(
						sNetId			:= 		gc_sADSNetID, 
						nSlaveAddr		:= 		gc_uiEP1908_EtherCATAdr, 
						nSubIndex		:= 		6, 
						nIndex			:= 		16#8003, 
						pDstBuf			:= 		ADR(wEP1908_VelLimit6), 
						cbBufLen		:= 		SIZEOF(wEP1908_VelLimit6), 
						bExecute		:= 		xExecute, 
						tTimeout		:= 		T#2S, 
						bBusy			=> 		xEP1908_VelLimit6_busy, 
						bError			=> 		xEP1908_VelLimit6_Err, 
						nErrId			=> 		udiEP1908_VelLimit6ID );

g_wHMI_EP1908_VelLimit6					:= 		wEP1908_VelLimit6 ;

iCaseVelLIMFiveScans := iCaseVelLIMFiveScans + 1 ; //Prevent code from passing through in only one pass

IF NOT xEP1908_VelLimit6_busy AND NOT xEP1908_VelLimit6_Err AND iCaseVelLIMFiveScans <> 0 THEN
	iFS_VelocityLimits := 6 ;
END_IF ;

6:
// EP1908-0002 FEATURES: Velocity Limit Channel 7
iCaseVelLIMFiveScans := 0 ;
fbEP1908_VelLimit7_EcCoESdoRead(
						sNetId			:= 		gc_sADSNetID, 
						nSlaveAddr		:= 		gc_uiEP1908_EtherCATAdr, 
						nSubIndex		:= 		7, 
						nIndex			:= 		16#8003, 
						pDstBuf			:= 		ADR(wEP1908_VelLimit7), 
						cbBufLen		:= 		SIZEOF(wEP1908_VelLimit7), 
						bExecute		:= 		xExecute, 
						tTimeout		:= 		T#2S, 
						bBusy			=> 		xEP1908_VelLimit7_busy, 
						bError			=> 		xEP1908_VelLimit7_Err, 
						nErrId			=> 		udiEP1908_VelLimit7ID );

g_wHMI_EP1908_VelLimit7					:= 		wEP1908_VelLimit7 ;

iCaseVelLIMSixScans := iCaseVelLIMSixScans + 1 ; //Prevent code from passing through in only one pass

IF NOT xEP1908_VelLimit7_busy AND NOT xEP1908_VelLimit7_Err AND iCaseVelLIMSixScans <> 0 THEN
	iFS_VelocityLimits := 7 ;
END_IF ;

7:
// EP1908-0002 FEATURES: Velocity Limit Channel 8
fbEP1908_VelLimit8_EcCoESdoRead(
						sNetId			:= 		gc_sADSNetID, 
						nSlaveAddr		:= 		gc_uiEP1908_EtherCATAdr, 
						nSubIndex		:= 		8, 
						nIndex			:= 		16#8003, 
						pDstBuf			:= 		ADR(wEP1908_VelLimit8), 
						cbBufLen		:= 		SIZEOF(wEP1908_VelLimit8), 
						bExecute		:= 		xExecute, 
						tTimeout		:= 		T#2S, 
						bBusy			=> 		xEP1908_VelLimit8_busy, 
						bError			=> 		xEP1908_VelLimit8_Err, 
						nErrId			=> 		udiEP1908_VelLimit8ID );

g_wHMI_EP1908_VelLimit8					:= 		wEP1908_VelLimit8 ;

iCaseVelLIMSevenScans := iCaseVelLIMSevenScans + 1 ; //Prevent code from passing through in only one pass

IF NOT xEP1908_VelLimit8_busy AND NOT xEP1908_VelLimit8_Err AND iCaseVelLIMSevenScans <> 0 THEN
	iFS_VelocityLimits := 0 ;
END_IF ;
	END_CASE ;

// Read the Primary Micro Controller (MC1) Temperature in DegC out of the EP1908-0002
IF C1.CV = 2 THEN
fbEP1908PriMCTemp_ADSRead(
						NETID			:= 		gc_sADSNetID, 
						PORT			:= 		gc_uiEP1908_EtherCATAdr, 
						IDXGRP			:= 		16#F302, 
						IDXOFFS			:= 		16#FA800001, 
						LEN				:= 		2, 
						DESTADDR		:= 		ADR(wEP1908_PriMCTemp), 
						READ			:= 		xExecute, 
						TMOUT			:= 		T#2S, 
						BUSY			=> 		xEP1908PriMCTemp_busy, 
						ERR				=> 		xEP1908PriMCTemp_Err, 
						ERRID			=> 		udiEP1908PriMCTemp_ErrID );

g_wHMI_EP1908PriMCTemp 						:= 		wEP1908_PriMCTemp ;
END_IF ;

// Read the Secondary Micro Controller (MC2) Temperature in DegC out of the EP1908-0002
IF C1.CV = 3 THEN
fbEP1908SecMCTemp_ADSRead(
						NETID			:= 		gc_sADSNetID, 
						PORT			:= 		gc_uiEP1908_EtherCATAdr, 
						IDXGRP			:= 		16#F302, 
						IDXOFFS			:= 		16#FA800002, 
						LEN				:= 		2, 
						DESTADDR		:= 		ADR(wEP1908_SecMCTemp), 
						READ			:= 		xExecute, 
						TMOUT			:= 		T#2S, 
						BUSY			=> 		xEP1908SecMCTemp_busy, 
						ERR				=> 		xEP1908SecMCTemp_Err, 
						ERRID			=> 		udiEP1908SecMCTemp_ErrID );

g_wHMI_EP1908SecMCTemp 						:= 		wEP1908_SecMCTemp ;
END_IF ;

// Read the Primary Micro Controller (MC1) Voltage in mV out of the EP1908-0002
IF C1.CV = 4 THEN
fbEP1908PriMCmV_ADSRead(
						NETID			:= 		gc_sADSNetID, 
						PORT			:= 		gc_uiEP1908_EtherCATAdr, 
						IDXGRP			:= 		16#F302, 
						IDXOFFS			:= 		16#FA810001, 
						LEN				:= 		2, 
						DESTADDR		:= 		ADR(wEP1908_PriMCmV), 
						READ			:= 		xExecute, 
						TMOUT			:= 		T#2S, 
						BUSY			=> 		xEP1908PriMCmV_busy, 
						ERR				=> 		xEP1908PriMCmV_Err, 
						ERRID			=> 		udiEP1908PriMCmV_ErrID );
						
g_wHMI_EP1908PriMC_Volts				:= 		WORD_TO_LREAL(wEP1908_PriMCmV) / 1000.0 ;
END_IF ;

// Read the Secondary Micro Controller (MC2) Voltage in mV out of the EP1908-0002
IF C1.CV = 5 THEN
fbEP1908SecMCmV_ADSRead(
						NETID			:= 		gc_sADSNetID, 
						PORT			:= 		gc_uiEP1908_EtherCATAdr, 
						IDXGRP			:= 		16#F302, 
						IDXOFFS			:= 		16#FA810002, 
						LEN				:= 		2, 
						DESTADDR		:= 		ADR(wEP1908_SecMCmV), 
						READ			:= 		xExecute, 
						TMOUT			:= 		T#2S, 
						BUSY			=> 		xEP1908SecMCmV_busy, 
						ERR				=> 		xEP1908SecMCmV_Err, 
						ERRID			=> 		udiEP1908SecMCmV_ErrID );
			
g_wHMI_EP1908SecMC_Volts 				:= 		WORD_TO_LREAL(wEP1908_SecMCmV) / 1000.0 ;
END_IF ;
	ELSE xReset := 1 ;
	END_IF ;
//
//		EP1908-0002 MODULE ALARMS
//
// EP1908-0002: Sensor Test Error
fbEP1908SensT_ADSRead(
						NETID			:= 		gc_sADSNetID, 
						PORT			:= 		gc_uiEP1908_EtherCATAdr, 
						IDXGRP			:= 		16#F302, 
						IDXOFFS			:= 		16#800E000A, 
						LEN				:= 		2, 
						DESTADDR		:= 		ADR(wEP1908_SenT), 
						READ			:= 		xExecute, 
						TMOUT			:= 		T#2S, 
						BUSY			=> 		xEP1908SenT_busy, 
						ERR				=> 		xEP1908SenT_Err, 
						ERRID			=> 		udiEP1908SenT_ErrID );

//These errors may only be present temporarily so they need to be latched and then cleared
//to be properly noted by the operator
g_xHMI_EP1908SenT1 						:= 		wEP1908_SenT.0 OR (g_xHMI_EP1908SenT1 AND NOT g_xHMI_EP1908_ErrClearPB) ;
g_xHMI_EP1908SenT2 						:= 		wEP1908_SenT.1 OR (g_xHMI_EP1908SenT2 AND NOT g_xHMI_EP1908_ErrClearPB) ;
g_xHMI_EP1908SenT3 						:= 		wEP1908_SenT.2 OR (g_xHMI_EP1908SenT3 AND NOT g_xHMI_EP1908_ErrClearPB) ;
g_xHMI_EP1908SenT4 						:= 		wEP1908_SenT.3 OR (g_xHMI_EP1908SenT4 AND NOT g_xHMI_EP1908_ErrClearPB) ;
g_xHMI_EP1908SenT5 						:= 		wEP1908_SenT.4 OR (g_xHMI_EP1908SenT5 AND NOT g_xHMI_EP1908_ErrClearPB) ;
g_xHMI_EP1908SenT6 						:= 		wEP1908_SenT.5 OR (g_xHMI_EP1908SenT6 AND NOT g_xHMI_EP1908_ErrClearPB) ;
g_xHMI_EP1908SenT7 						:= 		wEP1908_SenT.6 OR (g_xHMI_EP1908SenT7 AND NOT g_xHMI_EP1908_ErrClearPB) ;
g_xHMI_EP1908SenT8 						:= 		wEP1908_SenT.7 OR (g_xHMI_EP1908SenT8 AND NOT g_xHMI_EP1908_ErrClearPB) ;


// EP1908-002: 2-Channel Evaluation Error
// The two channels contradict each other (not same value)
fbEP1908_2CHEval_ADSRead(
						NETID			:= 		gc_sADSNetID, 
						PORT			:= 		gc_uiEP1908_EtherCATAdr, 
						IDXGRP			:= 		16#F302, 
						IDXOFFS			:= 		16#800E000B, 
						LEN				:= 		2, 
						DESTADDR		:= 		ADR(wEP1908_2CHEval), 
						READ			:= 		xExecute, 
						TMOUT			:= 		T#2S, 
						BUSY			=> 		xEP1908_2CHEval_busy, 
						ERR				=> 		xEP1908_2CHEval_Err, 
						ERRID			=> 		udiEP1908_2CHEval_ErrID );

//These errors may only be present temporarily so they need to be latched and then cleared
//to be properly noted by the operator
g_xHMI_EP1908_2CHEval_Pair1				:= 		wEP1908_2CHEval.0 OR (g_xHMI_EP1908_2CHEval_Pair1 AND NOT g_xHMI_EP1908_ErrClearPB) ;
g_xHMI_EP1908_2CHEval_Pair2				:= 		wEP1908_2CHEval.1 OR (g_xHMI_EP1908_2CHEval_Pair2 AND NOT g_xHMI_EP1908_ErrClearPB) ;
g_xHMI_EP1908_2CHEval_Pair3				:= 		wEP1908_2CHEval.2 OR (g_xHMI_EP1908_2CHEval_Pair3 AND NOT g_xHMI_EP1908_ErrClearPB) ;
g_xHMI_EP1908_2CHEval_Pair4				:= 		wEP1908_2CHEval.3 OR (g_xHMI_EP1908_2CHEval_Pair4 AND NOT g_xHMI_EP1908_ErrClearPB) ;


// EP1908-0002: Error In Safety Mat Operating Mode
// Input pairs not in the same state (not same value)
fbEP1908_SMiPair_ADSRead(
						NETID			:= 		gc_sADSNetID, 
						PORT			:= 		gc_uiEP1908_EtherCATAdr, 
						IDXGRP			:= 		16#F302, 
						IDXOFFS			:= 		16#800E000C, 
						LEN				:= 		2, 
						DESTADDR		:= 		ADR(wEP1908_SMiPair), 
						READ			:= 		xExecute, 
						TMOUT			:= 		T#2S, 
						BUSY			=> 		xEP1908_SMiPair_busy, 
						ERR				=> 		xEP1908_SMiPair_Err, 
						ERRID			=> 		udiEP1908_SMiPair_ErrID );

//These errors may only be present temporarily so they need to be latched and then cleared
//to be properly noted by the operator
g_xHMI_EP1908_SMiPair_Pair1				:= 		(wEP1908_SMiPair.0 AND wEP1908_SMiPair.1) OR (g_xHMI_EP1908_SMiPair_Pair1 AND NOT g_xHMI_EP1908_ErrClearPB) ;
g_xHMI_EP1908_SMiPair_Pair2				:= 		(wEP1908_SMiPair.2 AND wEP1908_SMiPair.3) OR (g_xHMI_EP1908_SMiPair_Pair2 AND NOT g_xHMI_EP1908_ErrClearPB) ;
g_xHMI_EP1908_SMiPair_Pair3				:= 		(wEP1908_SMiPair.4 AND wEP1908_SMiPair.5) OR (g_xHMI_EP1908_SMiPair_Pair3 AND NOT g_xHMI_EP1908_ErrClearPB) ;
g_xHMI_EP1908_SMiPair_Pair4				:= 		(wEP1908_SMiPair.6 AND wEP1908_SMiPair.7) OR (g_xHMI_EP1908_SMiPair_Pair4 AND NOT g_xHMI_EP1908_ErrClearPB) ;


// EP1908-0002: Error in Safety Mat Operating Supply
// External supply detected (Input channel not getting test pulses)
fbEP1908_SMExtSupply_ADSRead(
						NETID			:= 		gc_sADSNetID, 
						PORT			:= 		gc_uiEP1908_EtherCATAdr, 
						IDXGRP			:= 		16#F302, 
						IDXOFFS			:= 		16#800E000D, 
						LEN				:= 		2, 
						DESTADDR		:= 		ADR(wEP1908_SMExtSupply), 
						READ			:= 		xExecute, 
						TMOUT			:= 		T#2S, 
						BUSY			=> 		xEP1908_SMExtSupply_busy, 
						ERR				=> 		xEP1908_SMExtSupply_Err, 
						ERRID			=> 		udiEP1908_SMExtSupply_ErrID );

//These errors may only be present temporarily so they need to be latched and then cleared
//to be properly noted by the operator
g_xHMI_EP1908_SMExtSupply_CH1			:= 		wEP1908_SMExtSupply.0 OR (g_xHMI_EP1908_SMExtSupply_CH1 AND NOT g_xHMI_EP1908_ErrClearPB) ;
g_xHMI_EP1908_SMExtSupply_CH2			:= 		wEP1908_SMExtSupply.1 OR (g_xHMI_EP1908_SMExtSupply_CH2 AND NOT g_xHMI_EP1908_ErrClearPB) ;
g_xHMI_EP1908_SMExtSupply_CH3			:= 		wEP1908_SMExtSupply.2 OR (g_xHMI_EP1908_SMExtSupply_CH3 AND NOT g_xHMI_EP1908_ErrClearPB) ;
g_xHMI_EP1908_SMExtSupply_CH4			:= 		wEP1908_SMExtSupply.3 OR (g_xHMI_EP1908_SMExtSupply_CH4 AND NOT g_xHMI_EP1908_ErrClearPB) ;
g_xHMI_EP1908_SMExtSupply_CH5			:= 		wEP1908_SMExtSupply.4 OR (g_xHMI_EP1908_SMExtSupply_CH5 AND NOT g_xHMI_EP1908_ErrClearPB) ;
g_xHMI_EP1908_SMExtSupply_CH6			:= 		wEP1908_SMExtSupply.5 OR (g_xHMI_EP1908_SMExtSupply_CH6 AND NOT g_xHMI_EP1908_ErrClearPB) ;
g_xHMI_EP1908_SMExtSupply_CH7			:= 		wEP1908_SMExtSupply.6 OR (g_xHMI_EP1908_SMExtSupply_CH7 AND NOT g_xHMI_EP1908_ErrClearPB) ;
g_xHMI_EP1908_SMExtSupply_CH8			:= 		wEP1908_SMExtSupply.7 OR (g_xHMI_EP1908_SMExtSupply_CH8 AND NOT g_xHMI_EP1908_ErrClearPB) ;


// EP1908-0002: Error During Speed Monitoring
// Frquency Greater Than 500Hz
fbEP1908_FreqGT500_ADSRead(
						NETID			:= 		gc_sADSNetID, 
						PORT			:= 		gc_uiEP1908_EtherCATAdr, 
						IDXGRP			:= 		16#F302, 
						IDXOFFS			:= 		16#800E0013, 
						LEN				:= 		2, 
						DESTADDR		:= 		ADR(wEP1908_FreqGT500), 
						READ			:= 		xExecute, 
						TMOUT			:= 		T#2S, 
						BUSY			=> 		xEP1908_FreqGT500_busy, 
						ERR				=> 		xEP1908_FreqGT500_Err, 
						ERRID			=> 		udiEP1908_FreqGT500_ErrID );

//These errors may only be present temporarily so they need to be latched and then cleared
//to be properly noted by the operator
g_xHMI_EP1908_FreqGT500_CH1			:= 		wEP1908_FreqGT500.0 OR (g_xHMI_EP1908_FreqGT500_CH1 AND NOT g_xHMI_EP1908_ErrClearPB) ;
g_xHMI_EP1908_FreqGT500_CH2			:= 		wEP1908_FreqGT500.1 OR (g_xHMI_EP1908_FreqGT500_CH2 AND NOT g_xHMI_EP1908_ErrClearPB) ;
g_xHMI_EP1908_FreqGT500_CH3			:= 		wEP1908_FreqGT500.2 OR (g_xHMI_EP1908_FreqGT500_CH3 AND NOT g_xHMI_EP1908_ErrClearPB) ;
g_xHMI_EP1908_FreqGT500_CH4			:= 		wEP1908_FreqGT500.3 OR (g_xHMI_EP1908_FreqGT500_CH4 AND NOT g_xHMI_EP1908_ErrClearPB) ;
g_xHMI_EP1908_FreqGT500_CH5			:= 		wEP1908_FreqGT500.4 OR (g_xHMI_EP1908_FreqGT500_CH5 AND NOT g_xHMI_EP1908_ErrClearPB) ;
g_xHMI_EP1908_FreqGT500_CH6			:= 		wEP1908_FreqGT500.5 OR (g_xHMI_EP1908_FreqGT500_CH6 AND NOT g_xHMI_EP1908_ErrClearPB) ;
g_xHMI_EP1908_FreqGT500_CH7			:= 		wEP1908_FreqGT500.6 OR (g_xHMI_EP1908_FreqGT500_CH7 AND NOT g_xHMI_EP1908_ErrClearPB) ;
g_xHMI_EP1908_FreqGT500_CH8			:= 		wEP1908_FreqGT500.7 OR (g_xHMI_EP1908_FreqGT500_CH8 AND NOT g_xHMI_EP1908_ErrClearPB) ;


// EP1908-0002: Error In Operating Mode: Two Channel Sync Velocity Control
// Both inputs of a "pair" cannot be inactive in this mode
fbEP1908_BothInPairInact_ADSRead(
						NETID			:= 		gc_sADSNetID, 
						PORT			:= 		gc_uiEP1908_EtherCATAdr, 
						IDXGRP			:= 		16#F302, 
						IDXOFFS			:= 		16#800E0014, 
						LEN				:= 		2, 
						DESTADDR		:= 		ADR(wEP1908_BothInPairInact), 
						READ			:= 		xExecute, 
						TMOUT			:= 		T#2S, 
						BUSY			=> 		xEP1908_BothInPairInact_busy, 
						ERR				=> 		xEP1908_BothInPairInact_Err, 
						ERRID			=> 		udiEP1908_BothInPairInact_ErrID );

//These errors may only be present temporarily so they need to be latched and then cleared
//to be properly noted by the operator
g_xHMI_EP1908_BothInact_Pair1			:= 		wEP1908_BothInPairInact.0 OR (g_xHMI_EP1908_BothInact_Pair1 AND NOT g_xHMI_EP1908_ErrClearPB) ;
g_xHMI_EP1908_BothInact_Pair2			:= 		wEP1908_BothInPairInact.1 OR (g_xHMI_EP1908_BothInact_Pair2 AND NOT g_xHMI_EP1908_ErrClearPB) ;
g_xHMI_EP1908_BothInact_Pair3			:= 		wEP1908_BothInPairInact.2 OR (g_xHMI_EP1908_BothInact_Pair3 AND NOT g_xHMI_EP1908_ErrClearPB) ;
g_xHMI_EP1908_BothInact_Pair4			:= 		wEP1908_BothInPairInact.3 OR (g_xHMI_EP1908_BothInact_Pair4 AND NOT g_xHMI_EP1908_ErrClearPB) ;


// EP1908-0002: Error In Operating Modes: Two Channel Sync Velocity Control and Two Channel Encoder Velocity Control
// For a channel pair, two different motor speeds detected
fbEP1908_PairUnequalFreq_ADSRead(
						NETID			:= 		gc_sADSNetID, 
						PORT			:= 		gc_uiEP1908_EtherCATAdr, 
						IDXGRP			:= 		16#F302, 
						IDXOFFS			:= 		16#800E0015, 
						LEN				:= 		2, 
						DESTADDR		:= 		ADR(wEP1908_PairUnequalFreq), 
						READ			:= 		xExecute, 
						TMOUT			:= 		T#2S, 
						BUSY			=> 		xEP1908_PairUnequalFreq_busy, 
						ERR				=> 		xEP1908_PairUnequalFreq_Err, 
						ERRID			=> 		udiEP1908_PairUnequalFreq_ErrID );

//These errors may only be present temporarily so they need to be latched and then cleared
//to be properly noted by the operator
g_xHMI_EP1908_UnequalFreg_Pair1			:= 		wEP1908_PairUnequalFreq.0 OR (g_xHMI_EP1908_UnequalFreg_Pair1 AND NOT g_xHMI_EP1908_ErrClearPB) ;
g_xHMI_EP1908_UnequalFreg_Pair2			:= 		wEP1908_PairUnequalFreq.1 OR (g_xHMI_EP1908_UnequalFreg_Pair2 AND NOT g_xHMI_EP1908_ErrClearPB) ;
g_xHMI_EP1908_UnequalFreg_Pair3			:= 		wEP1908_PairUnequalFreq.2 OR (g_xHMI_EP1908_UnequalFreg_Pair3 AND NOT g_xHMI_EP1908_ErrClearPB) ;
g_xHMI_EP1908_UnequalFreg_Pair4			:= 		wEP1908_PairUnequalFreq.3 OR (g_xHMI_EP1908_UnequalFreg_Pair4 AND NOT g_xHMI_EP1908_ErrClearPB) ;


//Sum of all errors we know of in the EP1908 module
IF 		g_xHMI_EP1908SenT1 
	OR 	g_xHMI_EP1908SenT2 
	OR 	g_xHMI_EP1908SenT3 
	OR 	g_xHMI_EP1908SenT4
	OR 	g_xHMI_EP1908SenT5 
	OR 	g_xHMI_EP1908SenT6 
	OR 	g_xHMI_EP1908SenT7	
	OR 	g_xHMI_EP1908SenT8		
	OR 	g_xHMI_EP1908_2CHEval_Pair1	
	OR 	g_xHMI_EP1908_2CHEval_Pair2
	OR 	g_xHMI_EP1908_2CHEval_Pair3	
	OR 	g_xHMI_EP1908_2CHEval_Pair4	
	OR 	g_xHMI_EP1908_SMiPair_Pair1
	OR 	g_xHMI_EP1908_SMiPair_Pair2
	OR 	g_xHMI_EP1908_SMiPair_Pair3
	OR 	g_xHMI_EP1908_SMiPair_Pair4
	OR 	g_xHMI_EP1908_SMExtSupply_CH1
	OR 	g_xHMI_EP1908_SMExtSupply_CH2
	OR 	g_xHMI_EP1908_SMExtSupply_CH3
	OR 	g_xHMI_EP1908_SMExtSupply_CH4
	OR 	g_xHMI_EP1908_SMExtSupply_CH5
	OR 	g_xHMI_EP1908_SMExtSupply_CH6
	OR 	g_xHMI_EP1908_SMExtSupply_CH7
	OR 	g_xHMI_EP1908_SMExtSupply_CH8		
	OR 	g_xHMI_EP1908_FreqGT500_CH1
	OR 	g_xHMI_EP1908_FreqGT500_CH2
	OR 	g_xHMI_EP1908_FreqGT500_CH3
	OR 	g_xHMI_EP1908_FreqGT500_CH4
	OR 	g_xHMI_EP1908_FreqGT500_CH5
	OR 	g_xHMI_EP1908_FreqGT500_CH6
	OR 	g_xHMI_EP1908_FreqGT500_CH7
	OR 	g_xHMI_EP1908_FreqGT500_CH8
	OR 	g_xHMI_EP1908_BothInact_Pair1
	OR	g_xHMI_EP1908_BothInact_Pair2
	OR	g_xHMI_EP1908_BothInact_Pair3
	OR	g_xHMI_EP1908_BothInact_Pair4
	OR	g_xHMI_EP1908_UnequalFreg_Pair1
	OR	g_xHMI_EP1908_UnequalFreg_Pair2
	OR	g_xHMI_EP1908_UnequalFreg_Pair3
	OR	g_xHMI_EP1908_UnequalFreg_Pair4
THEN g_xHMI_EP1908_General_Error := TRUE ;
ELSE g_xHMI_EP1908_General_Error := FALSE ;
END_IF ;

END_PROGRAM

// ---- POUs/TwinSAFE_Function_Blocks_Info/FB_InfoDecoupler.TcPOU
FUNCTION_BLOCK FB_InfoDecoupler
VAR_INPUT
	stInfoData 			: 		DUT_ST_InfoDataFB ;
END_VAR
VAR_OUTPUT
	sState 				: 		STRING ;
END_VAR
VAR
END_VAR

// Decouple FB's State
IF stInfoData.usiMapState 			=	0 THEN
				sState 				:= 	'Undefined' ;
	ELSIF stInfoData.usiMapState 	= 	1 THEN
				sState 				:= 	'RUN' ;
	ELSIF stInfoData.usiMapState 	= 	2 THEN
				sState 				:= 	'STOP' ;
ELSE
				sState 				:= 	'Unknown' ;
END_IF

// The Decouple FB Has No Diagnostic Byte to Decode

END_FUNCTION_BLOCK

// ---- POUs/TwinSAFE_Function_Blocks_Info/FB_InfoMON.TcPOU
FUNCTION_BLOCK FB_InfoMON
VAR_INPUT
	stInfoData 			:		DUT_ST_InfoDataFB ;
END_VAR
VAR_OUTPUT
	sState 				: 		STRING ;
	sDiag 				: 		STRING ;
	END_VAR
VAR
END_VAR

// Guard Door Monitor FB's State
IF stInfoData.usiMapState 			= 	0 THEN
				sState 				:= 	'Undefined' ;
	ELSIF stInfoData.usiMapState 	= 	1 THEN
				sState 				:= 	'RUN' ;
	ELSIF stInfoData.usiMapState 	= 	2 THEN
				sState 				:= 	'STOP' ;
	ELSIF stInfoData.usiMapState 	= 	3 THEN
				sState 				:= 	'SAFE' ;
	ELSIF stInfoData.usiMapState 	= 	4 THEN
				sState 				:= 	'ERROR' ;
	ELSIF stInfoData.usiMapState 	= 	5 THEN
				sState 				:= 	'RESET' ;
	ELSIF stInfoData.usiMapState 	= 	6 THEN
				sState				:= 	'START' ;
	ELSIF stInfoData.usiMapState 	= 	7 THEN
				sState 				:= 	'Error Delay' ;
	ELSIF stInfoData.usiMapState 	= 	8 THEN
				sState 				:= 	'DelayOut' ;
	ELSIF stInfoData.usiMapState 	= 	9 THEN
				sState 				:= 	'Function Test' ;
	ELSE
				sState 				:= 	'Unknown' ;
END_IF

// Guard Door Monitor FB's Diagnostics
IF stInfoData.uiMapDiag 			= 	0 THEN
				sDiag 				:= 	'No Error' ;
ELSIF  stInfoData.uiMapDiag 		= 	1 THEN
				sDiag 				:= 	'Discrepancy Error of Input Group 1' ;
ELSIF  stInfoData.uiMapDiag 		= 	2 THEN
				sDiag 				:= 	'Discrepancy Error of Input Group 2' ;
ELSIF  stInfoData.uiMapDiag 		= 	4 THEN
				sDiag 				:= 	'Discrepancy Error of the Secure Inputs' ;
ELSIF  stInfoData.uiMapDiag 		= 	16 THEN
				sDiag 				:= 	'EDM 1 Monitoring Error' ;
ELSIF  stInfoData.uiMapDiag 		= 	32 THEN
				sDiag 				:= 	'EDM 2 Monitoring Error' ;
ELSE
				sDiag 				:= 	'Unknown' ;
END_IF

END_FUNCTION_BLOCK

// ---- POUs/TwinSAFE_Function_Blocks_Info/FB_InfoMuting.TcPOU
FUNCTION_BLOCK FB_InfoMuting
VAR_INPUT
	stInfoData 			:		DUT_ST_InfoDataFB ;
END_VAR
VAR_OUTPUT
	sState 				: 		STRING ;
	sDiag 				: 		STRING ;
	END_VAR
VAR
END_VAR

// Muting FB's State
IF stInfoData.usiMapState 			= 	0 THEN
				sState 				:= 	'Undefined' ;
	ELSIF stInfoData.usiMapState 	= 	1 THEN
				sState 				:= 	'RUN' ;
	ELSIF stInfoData.usiMapState 	= 	2 THEN
				sState 				:= 	'STOP' ;
	ELSIF stInfoData.usiMapState 	= 	3 THEN
				sState 				:= 	'SAFE' ;
	ELSIF stInfoData.usiMapState 	= 	4 THEN
				sState 				:= 	'ERROR' ;
	ELSIF stInfoData.usiMapState 	= 	5 THEN
				sState 				:= 	'RESET' ;
	ELSIF stInfoData.usiMapState 	= 	8 THEN
				sState 				:= 	'DelayOut' ;
	ELSIF stInfoData.usiMapState 	= 	9 THEN
				sState 				:= 	'Muting 1' ;
	ELSIF stInfoData.usiMapState	= 	10 THEN
				sState 				:= 	'Muting 2' ;
	ELSIF stInfoData.usiMapState 	= 	11 THEN
				sState 				:= 	'Muting 3' ;
	ELSIF stInfoData.usiMapState 	= 	12 THEN
				sState 				:= 	'Muting 4' ;
	ELSIF stInfoData.usiMapState 	= 	13 THEN
				sState 				:= 	'Muting 5' ;
	ELSIF stInfoData.usiMapState 	= 	14 THEN
				sState 				:= 	'Muting 6' ;
	ELSIF stInfoData.usiMapState 	= 	15 THEN
				sState 				:= 	'Muting 7' ;
	ELSIF stInfoData.usiMapState 	= 	16 THEN
				sState 				:= 	'Muting 8' ;
	ELSIF stInfoData.usiMapState 	= 	17 THEN
				sState 				:= 	'Muting 9' ;
	ELSE
				sState 				:= 	'Unknown' ;
END_IF

// Muting FB's Diagnostics
IF stInfoData.uiMapDiag 			= 	0 THEN
				sDiag 				:= 	'No Error' ;
ELSIF  stInfoData.uiMapDiag 		= 	1 THEN
				sDiag 				:= 	'Discrepancy Error In Muting Input Group 1' ;
ELSIF  stInfoData.uiMapDiag 		= 	2 THEN
				sDiag 				:= 	'Discrepancy Error In OSSD Input Group' ;
ELSIF  stInfoData.uiMapDiag 		= 	4 THEN
				sDiag 				:= 	'Discrepancy Error In Muting Input Group 2' ;
ELSIF  stInfoData.uiMapDiag 		= 	16 THEN
				sDiag 				:= 	'EDM 1 Monitoring Error' ;
ELSIF  stInfoData.uiMapDiag 		= 	32 THEN
				sDiag 				:= 	'EDM 2 Monitoring Error' ;
ELSIF  stInfoData.uiMapDiag 		= 	64 THEN
				sDiag 				:= 	'Muting Sequence Was Violated' ;
ELSIF  stInfoData.uiMapDiag 		= 	128 THEN
				sDiag 				:= 	'Maximum Muting Time Was Exceeded' ;
ELSE
				sDiag 				:= 	'Unknown' ;
END_IF

END_FUNCTION_BLOCK

// ---- POUs/TwinSAFE_Function_Blocks_Info/FB_InfoOperationMode.TcPOU
FUNCTION_BLOCK FB_InfoOperationMode
VAR_INPUT
	stInfoData 			:		DUT_ST_InfoDataFB ;
END_VAR
VAR_OUTPUT
	sState 				: 		STRING ;
	sDiag 				: 		STRING ;
	END_VAR
VAR
END_VAR

// Operating Mode FB's State
IF stInfoData.usiMapState 			= 	0 THEN
				sState 				:= 	'Undefined' ;
	ELSIF stInfoData.usiMapState 	= 	1 THEN
				sState 				:= 	'RUN' ;
	ELSIF stInfoData.usiMapState 	= 	2 THEN
				sState 				:= 	'STOP' ;
	ELSIF stInfoData.usiMapState 	= 	3 THEN
				sState 				:= 	'SAFE' ;
	ELSIF stInfoData.usiMapState 	= 	4 THEN
				sState 				:= 	'ERROR' ;
	ELSIF stInfoData.usiMapState 	= 	5 THEN
				sState 				:= 	'RESET' ;
	ELSIF stInfoData.usiMapState 	= 	6 THEN
				sState 				:= 	'START' ;
	ELSE
				sState 				:= 	'Unknown' ;
END_IF

// Operating Mode FB's Diagnostics
IF stInfoData.uiMapDiag 			= 	0 THEN
				sDiag 				:= 	'No Error' ;
ELSIF  stInfoData.uiMapDiag 		= 	1 THEN
				sDiag 				:= 	'Discrepancy Monitoring Error' ;
ELSE
				sDiag 				:= 	'Unknown' ;
END_IF

END_FUNCTION_BLOCK

// ---- POUs/TwinSAFE_Function_Blocks_Info/FB_InfoRS.TcPOU
FUNCTION_BLOCK FB_InfoRS
VAR_INPUT
	stInfoData 			: 		DUT_ST_InfoDataFB ;
END_VAR
VAR_OUTPUT
	sState 				: 		STRING ;
END_VAR
VAR
END_VAR

// RS FB's State
IF stInfoData.usiMapState 			= 	0 THEN
				sState 				:= 	'Undefined' ;
	ELSIF stInfoData.usiMapState 	= 	2 THEN
				sState 				:= 	'STOP' ;
	ELSIF stInfoData.usiMapState 	= 	3 THEN
				sState 				:= 	'SAFE' ;
	ELSIF stInfoData.usiMapState 	= 	9 THEN
				sState 				:= 	'SET' ;
	ELSE
				sState 				:= 	'Unknown' ;
END_IF

// The RS FB Has No Diagnostic Byte to Decode

END_FUNCTION_BLOCK

// ---- POUs/TwinSAFE_Function_Blocks_Info/FB_InfoSR.TcPOU
FUNCTION_BLOCK FB_InfoSR
VAR_INPUT
	stInfoData 			: 		DUT_ST_InfoDataFB ;
END_VAR
VAR_OUTPUT
	sState 				: 		STRING ;
END_VAR
VAR
END_VAR

// SR FB's State
IF stInfoData.usiMapState 			= 	0 THEN
				sState 				:= 	'Undefined' ;
	ELSIF stInfoData.usiMapState 	= 	2 THEN
				sState 				:= 	'STOP' ;
	ELSIF stInfoData.usiMapState 	= 	3 THEN
				sState 				:= 	'SAFE' ;
	ELSIF stInfoData.usiMapState 	= 	9 THEN
				sState 				:= 	'SET' ;
	ELSE
				sState 				:= 	'Unknown' ;
END_IF

// The SR FB Has No Diagnostic Byte to Decode

END_FUNCTION_BLOCK

